Yaskawa INFORM job: X4-SCHODKI_ZEW_HARDOX.JBI

/JOB
//NAME X4-SCHODKI_ZEW_HARDOX
//POS
///NPOS 533,533,533,13,0,0
///TOOL 0
///POSTYPE PULSE
///PULSE
C00000=-21160,-126487,-99095,-6220,53097,-19917
C00001=-122314,-84956,-84267,-5758,65294,-20346
C00002=-113867,-2788,-32259,-11364,77586,20622
C00003=-111699,9606,-11794,-12514,71800,21939
C00004=-110873,16102,-4909,-12893,71047,22311
C00005=-111426,18220,-2948,-12689,70847,22135
C00006=-111334,17863,-3281,-12723,70881,22164
C00007=-111334,17842,-1921,-12786,70054,22254
C00008=-111688,13758,-7042,-12574,71029,22022
C00009=-137921,23655,2193,26065,80546,-13065
C00010=-138187,30095,8478,26164,80127,-13260
C00011=-137141,31636,10013,25924,79665,-12972
C00012=-137283,31426,9804,25956,79727,-13011
C00013=-137283,31447,11085,26011,79025,-13166
C00014=-137811,24810,3269,26040,80453,-13045
C00015=-130093,15204,-5597,17076,73087,-3422
C00016=-130254,16762,-4164,17139,73044,-3486
C00017=-130499,11823,-8660,17205,73314,-3535
C00018=-136657,16032,-4835,19303,74485,-5576
C00019=-136779,34044,12201,19450,73350,-5806
C00020=-136367,37287,16065,19383,72578,-5782
C00021=-135529,38270,17077,19116,72272,-5524
C00022=-135735,38345,17156,19186,72312,-5593
C00023=-135735,38391,18179,19247,71738,-5687
C00024=-136093,38073,17157,19317,72259,-5733
C00025=-136821,38987,18103,19565,72324,-5991
C00026=-137234,41236,20445,19732,72152,-6174
C00027=-137468,37941,16529,19737,72884,-6137
C00028=-139273,33119,8814,10616,74138,-14432
C00029=-138400,39162,15428,10360,73077,-14220
C00030=-137624,40756,17090,10099,72782,-13973
C00031=-137810,40443,16764,10163,72844,-14033
C00032=-137810,40460,18419,10216,71849,-14119
C00033=-138377,33107,10032,10341,73283,-14197
C00034=-129933,32626,9546,-1459,71562,-3103
C00035=-130107,34413,11352,-1398,71367,-3162
C00036=-130344,28976,5916,-1305,71915,-3250
C00037=-134876,30968,7890,396,71698,-4822
C00038=-142592,70732,50995,12851,68399,-16892
C00039=-141830,71409,51797,12602,68137,-16639
C00040=-142006,70894,51186,12652,68274,-16689
C00041=-142006,71149,52557,12712,67578,-16765
C00042=-142006,71007,51815,12679,67954,-16725
C00043=-142747,76515,58410,13043,66871,-17119
C00044=-142702,66110,44987,12780,69711,-16790
C00045=-130401,22900,-3912,-9781,74013,-14096
C00046=-130750,-77898,-76934,-10038,67211,-13654
C00047=-128341,-94500,-64478,-15665,37561,-8814
C00048=-125354,-34494,-33676,-16070,41961,-8103
C00049=-123908,-22688,-35224,7311,60763,-8117
C00050=-115329,1774,-22996,8583,68206,-33205
C00051=-113811,6923,-16554,7934,66753,-32769
C00052=-112938,8598,-15088,7517,66630,-32466
C00053=-113357,7607,-15958,7718,66694,-32611
C00054=-113357,7474,-14642,7767,65823,-32669
C00055=-113357,7562,-15559,7732,66427,-32629
C00056=-114674,8046,-17033,9196,71995,-10105
C00057=-114277,9137,-16073,9034,71921,-9973
C00058=-114994,10710,-14679,9331,71949,-10219
C00059=-115929,5782,-19714,10610,72890,-11247
C00060=-114914,9168,-18033,20160,83408,-25507
C00061=-115077,46309,11834,20851,92481,-23935
C00062=-115077,45981,13257,20825,91503,-24106
C00063=-115077,46309,11834,20851,92481,-23935
C00064=-114509,10430,-16126,20066,82816,-25464
C00065=-113574,12027,-14696,19812,82540,-25184
C00066=-113966,9476,-16971,19916,82715,-25292
C00067=-109617,50730,10299,20838,92897,-21763
C00068=-109849,50897,10058,15384,88802,-23804
C00069=-109890,48745,8449,15106,86687,-24128
C00070=-110280,52401,12404,10304,83703,-19954
C00071=-110340,48514,8983,10012,81065,-20250
C00072=-109875,50139,10594,6927,80049,-17487
C00073=-111642,41129,-2073,7513,83338,-17864
C00074=-120740,-4591,-30289,15267,55452,-23675
C00075=-120758,-111403,-89341,20679,37744,-27189
C00076=-120758,-111403,-89341,20679,37744,-27189
C00077=-97140,-41370,-74515,-11864,90116,15742
C00078=-93918,-16818,-51601,-15265,90472,19448
C00079=-96838,-21310,-54909,-14446,89719,18600
C00080=-97144,-22320,-55662,-14359,89616,18514
C00081=-98771,-24881,-57497,-13895,89173,18041
C00082=-115828,-29996,-61044,7286,86100,-2495
C00083=-121364,-24267,-57094,13933,89260,-9154
C00084=-125064,-13370,-49143,14990,90552,-10191
C00085=-125209,-12228,-48362,15033,90681,-10222
C00086=-127775,-3453,-41245,15747,91251,-10973
C00087=-117906,-11103,-47413,1372,86513,3179
C00088=-107817,-4833,-42392,-13913,90158,17947
C00089=-111065,-8601,-45456,-12965,89620,16971
C00090=-111228,-9142,-45834,-12917,89553,16926
C00091=-113235,-11504,-47787,-12324,89257,16321
C00092=-116129,-16038,-53218,-11461,89860,15351
C00093=-132129,3503,-37461,-731,88042,5165
C00094=-135089,9999,-29918,1559,86605,3002
C00095=-133932,10352,-29664,1179,86614,3356
C00096=-133300,11122,-28999,967,86593,3553
C00097=-132997,13157,-27039,5636,86965,-851
C00098=-131112,-12606,-50888,7793,88905,-29033
C00099=-129834,-10886,-48018,7386,87922,-28697
C00100=-133242,1411,-38107,8469,88444,-29724
C00101=-133268,2556,-37251,8479,88508,-29727
C00102=-132895,14601,-26523,2898,86979,-24450
C00103=-133144,15447,-25750,2979,86944,-24527
C00104=-133588,9909,-35564,3125,90148,-24585
C00105=-114600,-38617,-66572,-24501,76796,-21744
C00106=-88804,-102668,-113384,-34072,81784,-13502
C00107=3643,-76224,-106676,19950,71810,76872
C00108=6047,-95755,-92046,-14751,98253,9605
C00109=8024,-164446,-133802,-16041,6272,12396
C00110=8024,-164446,-133802,-16041,6272,12396
C00111=80911,-131071,-112390,-19160,57527,-4768
C00112=107387,-112645,-89313,-18613,48039,-3448
C00113=120529,-94925,-67119,-18087,38914,-2179
C00114=119158,-22093,-21003,-8683,62714,-5793
C00115=120616,-13235,-11129,-9376,61371,-5124
C00116=120244,-10241,-8815,-9223,61441,-5272
C00117=120242,-11093,-9478,-9225,61411,-5270
C00118=120242,-10458,-7028,-9331,60244,-5174
C00119=120224,-17007,-14555,-9215,61493,-5286
C00120=122889,-18524,910,-53470,54044,-6110
C00121=122847,-15690,3005,-53366,54123,-6195
C00122=122811,-12986,5045,-53281,54183,-6262
C00123=122821,-13724,4484,-53302,54168,-6245
C00124=122821,-12957,6355,-53740,53705,-5906
C00125=125895,-21581,-2992,-53539,56263,-5738
C00126=123923,-36868,-26996,-37261,61302,-5894
C00127=108816,-52753,-53811,-10212,62008,-9374
C00128=96034,-45136,-47055,9675,61622,-25160
C00129=97205,-43220,-45890,9111,61748,-24699
C00130=96974,-43470,-46044,9221,61740,-24787
C00131=96974,-43222,-44278,9303,60791,-24865
C00132=96448,-45521,-47615,9470,61714,-24990
C00133=118629,-40101,-48504,-12157,74776,12413
C00134=119364,-34097,-44083,-12359,75244,12623
C00135=118100,-32224,-42841,-11965,75251,12181
C00136=118253,-32582,-43080,-12015,75236,12237
C00137=118253,-32540,-41664,-12057,74406,12319
C00138=118721,-32602,-42752,-12165,75101,12411
C00139=116137,-37716,-46090,-11401,74165,11593
C00140=108993,-39238,-47060,-3979,71836,3847
C00141=109761,-37600,-46019,-4238,72074,4108
C00142=108993,-39238,-47060,-3979,71836,3847
C00143=117414,-43467,-49690,-6866,71847,6805
C00144=120406,-23125,-36428,-7781,74390,7697
C00145=120412,-21128,-34805,-7781,74419,7698
C00146=119620,-19753,-33804,-7516,74437,7425
C00147=119849,-20298,-34202,-7592,74423,7506
C00148=119849,-20300,-33096,-7616,73750,7551
C00149=119849,-20302,-33703,-7602,74119,7528
C00150=120845,-19874,-33391,-7929,74241,7866
C00151=121446,-18122,-32105,-8123,74405,8066
C00152=121464,-22241,-35587,-8130,74432,8070
C00153=122270,-32243,-42159,4732,69932,24573
C00154=121378,-24903,-37120,5049,70656,24286
C00155=120376,-23507,-36128,5424,70830,23939
C00156=120533,-24190,-36613,5366,70768,23993
C00157=120533,-24175,-35602,5386,70155,23966
C00158=120148,-30314,-42064,5504,71001,23867
C00159=110805,-25383,-38662,15109,74916,14576
C00160=111818,-22665,-36734,14771,74934,14940
C00161=111748,-27369,-40047,14817,74581,14871
C00162=119775,-28434,-40781,12151,73173,17551
C00163=124224,-1084,-19915,10540,73751,19166
C00164=130157,198,-18683,-209,73628,24476
C00165=130157,158,-17341,-210,72780,24477
C00166=130157,185,-18394,-210,73442,24477
C00167=129196,1421,-17357,132,73439,24146
C00168=130157,185,-18394,-210,73442,24477
C00169=122787,3680,-15441,12656,76349,11624
C00170=123743,5439,-13926,12357,76179,11938
C00171=123109,1410,-18093,12531,76759,11776
C00172=126751,-18741,-32489,13679,66636,29547
C00173=131594,-6512,-22252,11541,65879,31250
C00174=135627,-1986,-17513,3780,65616,32121
C00175=134567,7692,-12619,5089,73681,32152
C00176=134567,7658,-11680,5104,73087,32127
C00177=135627,-1986,-17486,3780,65599,32120
C00178=134800,-891,-16582,4152,65645,31822
C00179=135627,-1986,-17486,3780,65599,32120
C00180=122949,-12611,-24589,22132,67603,15841
C00181=121506,-8744,-21577,22663,68115,15387
C00182=122081,-6475,-19773,22437,68011,15585
C00183=121506,-8744,-21577,22663,68115,15387
C00184=127706,-12999,-26066,20142,67056,17565
C00185=135610,17691,-1290,8706,67320,35420
C00186=135610,17711,-348,8741,66754,35378
C00187=136075,11798,-4304,8086,62236,35152
C00188=136366,13707,-2741,6760,62424,35173
C00189=136075,11798,-4304,8086,62236,35152
C00190=131305,-10305,-23416,10361,63176,33430
C00191=168291,-111367,-82610,-9688,47305,48503
C00192=206286,-74639,-65979,-25452,64014,61826
C00193=159660,-110455,-93035,-14572,38895,45711
C00194=139772,-9678,-45421,-20416,66544,-77404
C00195=128522,-26109,-48700,-36268,57340,-84657
C00196=119767,-9340,-33749,-20588,54929,-87055
C00197=118381,-12869,-36453,-19680,54464,-87541
C00198=118069,-13852,-36761,-19540,54093,-87599
C00199=119937,-17804,-39758,-30591,59034,-81437
C00200=119898,-18805,-40392,-30604,58911,-81418
C00201=117451,-25827,-45422,-31757,59099,-80707
C00202=119398,-27349,-44114,-37266,57847,-80053
C00203=122977,-25509,-47564,-34287,62428,-79397
C00204=137466,-21144,-46854,-40649,69913,-75869
C00205=196853,-39310,-56838,-56279,98183,-62272
C00206=239125,-37728,-55833,-56309,98295,-62347
C00207=198880,-64017,-70083,-47949,71692,22240
C00208=95782,-63494,-66422,9583,64100,-25040
C00209=96608,-32442,-40990,7123,69750,-24476
C00210=99153,-41436,-44893,7278,64322,-23821
C00211=98934,-42045,-45261,7777,64334,-23890
C00212=100370,-44106,-46526,7182,63922,-23380
C00213=119741,-40174,-44096,-19149,69535,-259
C00214=121592,-27553,-38534,-18093,79240,10876
C00215=125227,-17250,-31142,-18927,80757,11935
C00216=125393,-15914,-30142,-18963,80861,11977
C00217=127846,-8061,-24015,-19516,81680,12716
C00218=119795,-17677,-31449,-8017,74335,-710
C00219=108325,-15786,-29976,9492,74890,-18554
C00220=111630,-19800,-33189,8434,74445,-17438
C00221=111755,-20573,-33754,8397,74383,-17399
C00222=113687,-22438,-34957,7772,73974,-16756
C00223=117056,-24250,-37509,6639,74313,-15568
C00224=128480,-979,-19969,3779,76440,-7427
C00225=130214,3282,-15364,3237,75722,-6858
C00226=129537,3735,-15090,2864,75741,-6451
C00227=129186,4471,-14460,2975,75747,-6572
C00228=129576,5579,-13546,-2876,75741,-370
C00229=130057,-3886,-22978,-3018,76699,-230
C00230=122913,-28792,-41505,-1480,73376,7564
C00231=125274,-18849,-33719,-4896,77191,17730
C00232=131975,-10313,-25549,-10610,74903,19808
C00233=132069,-9167,-24748,-10635,75011,19832
C00234=135966,6668,-11544,-11862,75556,21141
C00235=130236,2592,-15119,-2350,73160,11427
C00236=128403,-11609,-30449,-1692,75251,10764
C00237=112588,-48510,-57222,11111,73491,6010
C00238=118900,-27089,-23855,-4947,60648,-6067
C00239=130292,-938,239,-22775,68727,4409
C00240=117379,-19874,-3208,-40401,48526,-8648
C00241=111452,-18537,-670,-42583,47269,-4687
C00242=115600,-23691,-9256,-36668,53200,-7502
C00243=123114,-34014,-31898,-14023,63529,-7414
C00244=103776,-61917,-65189,16989,73535,3120
C00245=77625,-115928,-93453,24842,70557,-7280
C00246=80911,-131071,-112390,-19160,57527,-4768
C00247=8024,-164446,-133802,-16041,6272,12396
C00248=8024,-164446,-133802,-16041,6272,12396
C00249=3643,-76224,-106676,19950,71810,76872
C00250=3643,-76224,-106676,19950,71810,76872
C00251=3643,-76224,-106676,19950,71810,76872
C00252=3643,-76224,-106676,19950,71810,76872
C00253=-84926,-80067,-84751,-11816,58952,90735
C00254=-123661,-80067,-84751,-11816,58952,90735
C00255=-122903,-30976,-67088,-11139,71240,89773
C00256=-127139,198,-37668,-8934,68706,88593
C00257=-128438,61784,5096,-11296,104956,84706
C00258=-128499,61338,5461,-11257,104502,84732
C00259=-128499,60609,6014,-11216,103801,84798
C00260=-128499,60703,5938,-11219,103891,84788
C00261=-128273,58374,3262,-11283,104361,84815
C00262=-129063,60229,5392,-11127,103914,84609
C00263=-129975,59592,4657,-10979,103923,84320
C00264=-129063,61136,4723,-11178,104777,84528
C00265=-133608,25580,-26809,3658,85338,86524
C00266=-133451,25659,-25652,3594,84661,86550
C00267=-133451,25176,-25219,3596,84144,86535
C00268=-133451,25290,-25323,3596,84268,86539
C00269=-133704,27427,-23228,3702,84086,86458
C00270=-132883,25504,-25115,3358,84228,86706
C00271=-131959,26058,-24571,2972,84149,86977
C00272=-132883,26390,-25891,3354,85159,86731
C00273=-124009,23376,-33099,9871,93491,73495
C00274=-123836,21523,-31842,9785,91773,73411
C00275=-123836,21007,-31440,9780,91267,73370
C00276=-123836,21118,-31523,9779,91378,73378
C00277=-124020,21136,-31509,9844,91394,73325
C00278=-123836,21717,-31986,9786,91960,73425
C00279=-123362,54647,1396,9599,88337,73286
C00280=-123280,54093,1879,9571,87758,73266
C00281=-123280,53580,2373,9572,87197,73224
C00282=-123280,53684,2271,9572,87311,73232
C00283=-123445,53701,2290,9630,87327,73184
C00284=-123280,54390,1609,9571,88071,73290
C00285=-125487,1894,-47010,15546,81241,73431
C00286=-125038,-918,-46164,15415,79269,73319
C00287=-125038,-1557,-45483,15449,78547,73228
C00288=-125038,-1296,-45768,15435,78846,73266
C00289=-124792,-4958,-48763,15321,78767,73334
C00290=-124792,-5291,-48397,15341,78383,73286
C00291=-124942,-3860,-47236,15411,78431,73246
C00292=-124949,-3247,-48411,15367,79433,73371
C00293=-117766,4954,-42293,11937,78807,75522
C00294=-117765,4385,-41727,11960,78179,75462
C00295=-117765,3691,-40987,11993,77383,75384
C00296=-117765,3905,-41223,11983,77632,75409
C00297=-117315,-1199,-45523,11766,77597,75546
C00298=-117315,-1510,-45179,11782,77233,75510
C00299=-117558,529,-43483,11899,77268,75437
C00300=-117512,138,-43810,11877,77262,75451
C00301=-118420,-299,-44174,12317,77382,75178
C00302=-118236,775,-45287,12178,78567,75353
C00303=-118072,3935,-47958,-6388,83076,70255
C00304=-117672,-3023,-48934,-6614,80148,70526
C00305=-117672,-3736,-48216,-6630,79346,70569
C00306=-117672,-3529,-48430,-6626,79583,70556
C00307=-117228,-8786,-52641,-6836,79506,70694
C00308=-117228,-9038,-52379,-6842,79217,70710
C00309=-117506,-6503,-50372,-6711,79263,70623
C00310=-117501,-5841,-51500,-6695,80291,70569
C00311=-140420,-5323,-52894,-1425,79407,62151
C00312=-145152,-6893,-50667,901,77218,60735
C00313=-145152,-7520,-49981,903,76471,60731
C00314=-145152,-7282,-50248,902,76758,60733
C00315=-145549,-12922,-54644,1100,76568,60610
C00316=-145549,-13251,-54270,1101,76169,60607
C00317=-145357,-10860,-52432,1005,76265,60667
C00318=-145454,-10428,-54083,1049,77503,60647
C00319=-128438,61784,5096,-11296,104956,84706
C00320=-125432,64694,8496,-11765,104746,85676
C00321=-124662,61530,7092,-11845,104102,85987
C00322=-129042,57667,2638,-11155,104293,84576
C00323=-129042,57667,2638,-11155,104293,84576
C00324=-130604,43844,-10848,-9440,96834,84970
C00325=-134320,25640,-25171,-1592,84682,85843
C00326=-137130,19028,-28909,5529,79562,86298
C00327=-133173,20661,-27367,3689,79252,87491
C00328=-133173,20661,-27367,3689,79252,87491
C00329=-130137,46597,-8299,-623,96129,87922
C00330=-124662,61530,7092,-11845,104102,85987
C00331=-124774,62733,6607,-11885,104986,85864
C00332=-124009,23376,-33099,9871,93491,73495
C00333=-124132,1653,-46107,10219,82838,72685
C00334=-124081,891,-45397,10214,82014,72632
C00335=-123957,9856,-37642,10163,81837,72656
C00336=-123957,10397,-38161,10152,82425,72704
C00337=-123328,56859,331,9544,106484,74564
C00338=-123371,55361,-743,9544,106381,74542
C00339=-123850,18974,-31534,9940,86065,72993
C00340=-123271,52328,2620,9755,82174,72867
C00341=-123271,52662,2260,9748,82562,72897
C00342=-127589,85070,34886,10208,94705,72346
C00343=-127605,84117,34810,10205,94272,72304
C00344=-128402,52886,4535,12032,80236,71108
C00345=-128225,58749,11133,11991,79186,71062
C00346=-128225,59756,9915,11950,80426,71182
C00347=-127948,-6468,-52224,16731,80618,72590
C00348=-127424,-2906,-46525,16565,78913,72521
C00349=-130398,-3517,-45707,22203,78529,72642
C00350=-129750,-4200,-46262,21908,78366,72825
C00351=-128378,-4058,-46148,21277,78045,73219
C00352=-121663,-2339,-44741,18114,76618,75175
C00353=-115640,-347,-45187,7560,78187,75189
C00354=-115728,877,-44163,7601,78193,75162
C00355=-120769,-437,-43402,17007,76693,75297
C00356=-117743,897,-42286,15536,76152,76198
C00357=-117743,1848,-43354,15471,77259,76340
C00358=-127948,-6468,-52224,16731,80618,72590
C00359=-117890,-3178,-50858,3,81161,72238
C00360=-118337,-2948,-47894,214,79455,72104
C00361=-118633,-4108,-48842,352,79442,72013
C00362=-119043,-4814,-49224,544,79316,71888
C00363=-117595,-6540,-50048,-6610,79040,70621
C00364=-148660,-7034,-50440,8059,79279,61212
C00365=-144502,-3981,-44897,-14956,77034,56051
C00366=-144502,-3024,-46070,-14896,78209,55905
C00367=-121650,-5019,-58113,-24818,88994,61227
C00368=-122271,-90655,-108273,-25102,76857,63579
C00369=32571,-155976,-119807,-12475,-16322,90735
C00370=32571,-155976,-119807,-12475,-16322,90735
C00371=432,-155976,-119807,-12475,-16322,90735
C00372=432,-155976,-119807,609,74424,82099
C00373=109557,-155976,-119807,609,74424,82099
C00374=131526,-73725,-103845,608,74936,82102
C00375=123676,15402,-35905,4513,79152,79802
C00376=123062,13907,-34117,4846,77322,79548
C00377=123062,13234,-33422,4858,76552,79519
C00378=123062,13371,-33570,4856,76713,79525
C00379=122641,9174,-37336,5063,76896,79403
C00380=122641,8998,-37151,5067,76691,79395
C00381=122935,11565,-34861,4920,76586,79481
C00382=122946,11968,-36957,4889,78077,79544
C00383=128447,74843,20112,4181,96979,82150
C00384=125283,85916,34561,10572,99934,82307
C00385=125283,85252,35263,10543,99176,82240
C00386=125283,85360,35146,10549,99299,82250
C00387=125053,82619,31732,10612,100007,82237
C00388=130133,63218,10337,-478,91768,81983
C00389=129424,63758,10966,-266,91655,81768
C00390=130133,64176,9529,-479,92758,81979
C00391=130562,33088,-16638,4936,77416,83764
C00392=130793,32566,-15857,4835,76660,83805
C00393=130793,32167,-15406,4840,76179,83784
C00394=130793,32267,-15524,4840,76302,83790
C00395=131028,34733,-13015,4729,76015,83854
C00396=131220,32098,-15696,4631,76299,83921
C00397=132054,31571,-16260,4222,76334,84182
C00398=131220,33089,-16758,4612,77459,83964
C00399=139932,37494,-12236,353,76701,86621
C00400=140087,35879,-12490,279,76027,86666
C00401=140087,35493,-12044,279,75554,86665
C00402=140087,35594,-12164,279,75679,86665
C00403=140066,35120,-12650,289,75735,86658
C00404=140191,35640,-13057,228,76251,86698
C00405=144017,27791,-20964,-1648,77113,87870
C00406=144452,26542,-22051,-1859,77149,88000
C00407=144452,26082,-21554,-1861,76609,88006
C00408=144452,26191,-21674,-1860,76739,88004
C00409=144404,25656,-22195,-1836,76786,87989
C00410=144440,26768,-22186,-1850,77351,87992
C00411=131883,61278,7206,30840,98791,74831
C00412=134379,62597,12993,30002,95475,74827
C00413=134379,61982,13733,29953,94803,74651
C00414=134379,62041,13659,29957,94869,74668
C00415=134641,60677,12085,29912,95014,74800
C00416=134557,61287,11866,29960,95432,74879
C00417=135751,64817,15957,29630,94430,75042
C00418=135751,64366,16527,29599,93921,74910
C00419=135751,64464,16397,29606,94034,74940
C00420=136038,63706,15517,29546,94076,75054
C00421=135884,64035,14878,29615,94618,75138
C00422=132248,54311,3772,30620,97400,74580
C00423=132248,53898,4219,30579,96978,74466
C00424=132248,54015,4093,30592,97096,74498
C00425=129743,23890,-20564,36987,85720,58400
C00426=129743,23766,-20396,36992,85584,58355
C00427=129558,27733,-16530,37067,85382,58218
C00428=129612,27679,-19165,37009,86646,58668
C00429=128447,74843,20112,4181,96979,82150
C00430=123342,73095,22025,-160,83462,78859
C00431=123154,73616,24314,-89,82322,78803
C00432=123153,73142,24904,-89,81719,78803
C00433=123153,73214,24808,-89,81815,78803
C00434=123322,73233,24831,-152,81812,78855
C00435=123242,73796,24123,-122,82537,78829
C00436=123688,38124,-16975,-287,89497,78950
C00437=123584,37405,-16446,-248,88799,78920
C00438=123584,36852,-15992,-248,88235,78921
C00439=123584,36953,-16076,-248,88338,78921
C00440=123771,37027,-15999,-318,88331,78976
C00441=123711,37942,-16737,-296,89256,78956
C00442=125600,30882,-21833,-7436,86676,77848
C00443=125600,30421,-21439,-7437,86203,77876
C00444=125600,30651,-21637,-7436,86441,77862
C00445=125408,25580,-26659,-7358,86908,77778
C00446=125408,25321,-26441,-7359,86643,77794
C00447=125473,27805,-24002,-7386,86425,77827
C00448=125473,28768,-24793,-7383,87400,77770
C00449=119735,35798,-17668,-5085,86249,76136
C00450=119539,34421,-18220,-5006,85875,76095
C00451=119539,33880,-17746,-5008,85308,76118
C00452=119539,34054,-17902,-5007,85493,76110
C00453=119038,29010,-22988,-4803,86002,75940
C00454=119038,28800,-22804,-4803,85784,75950
C00455=119400,31604,-19998,-4950,85517,76067
C00456=119348,31196,-20409,-4929,85557,76050
C00457=119987,30698,-20909,-5185,85643,76236
C00458=119878,31262,-21389,-5139,86220,76180
C00459=128447,74843,20112,4181,96979,82150
C00460=124116,94593,46679,11672,102200,82046
C00461=127992,89556,40269,11396,103012,83415
C00462=127992,89556,40269,11396,103012,83415
C00463=129587,64527,11769,9334,94236,82902
C00464=132949,55867,3405,1789,88718,82304
C00465=135017,42183,-7617,-3983,80598,81730
C00466=131389,44285,-5377,-2395,80172,80630
C00467=131389,44285,-5377,-2395,80172,80630
C00468=132236,58768,6599,-5557,89172,80111
C00469=124116,94593,46679,11672,102200,82046
C00470=124104,96699,46972,11722,103085,82128
C00471=143616,55927,3157,-10764,85977,88488
C00472=148648,52226,4712,-20280,79209,89000
C00473=148516,52517,6145,-20267,78491,89078
C00474=148493,50806,4254,-20239,78754,89026
C00475=148493,50806,4254,-20239,78754,89026
C00476=140540,62715,11224,-1744,88121,79582
C00477=136875,97884,50516,6622,100207,80085
C00478=137178,101903,55708,7300,101861,80376
C00479=141388,85873,34619,7196,106210,82037
C00480=141388,85873,34619,7196,106210,82037
C00481=144251,72599,18557,4985,103495,82483
C00482=142808,65433,11761,11663,99026,82997
C00483=143036,65995,12421,11611,98881,83056
C00484=141225,66295,15146,18784,94862,83443
C00485=141225,67539,13983,18842,96148,83643
C00486=134946,24098,-37413,1605,94871,78009
C00487=119914,5828,-43406,7387,78039,72896
C00488=119947,11480,-35472,7422,76073,72788
C00489=122612,12239,-33354,1270,74705,81494
C00490=122593,20325,-25822,1280,74225,81483
C00491=122593,20926,-26500,1276,74951,81491
C00492=122252,68374,13418,1881,98899,81800
C00493=122183,71569,17944,1970,100800,81820
C00494=122504,26900,-20597,1350,76261,81486
C00495=122262,60388,15081,1504,71520,81353
C00496=122262,60839,14399,1498,72171,81361
C00497=122138,113341,70542,1866,86603,81577
C00498=122006,122876,83892,1956,86819,81545
C00499=122146,80790,34625,1654,78685,81435
C00500=122106,87009,42344,1679,77132,81400
C00501=122106,87849,40937,1672,78429,81417
C00502=119914,5828,-43406,7387,78039,72896
C00503=119947,11480,-35472,7422,76073,72788
C00504=127628,12770,-32579,-8395,74956,81127
C00505=127315,11373,-33838,-8234,74983,81029
C00506=128071,4553,-37059,-10767,69794,81127
C00507=127715,4566,-37046,-10566,69753,81013
C00508=126468,4857,-36794,-9866,69606,80617
C00509=120231,6674,-35162,-6323,68971,78621
C00510=109035,9040,-32856,15253,70226,79190
C00511=109194,10411,-31638,15171,70156,79234
C00512=119176,8835,-33361,-5116,68948,78440
C00513=122835,8933,-31103,-15912,67286,77485
C00514=123391,8334,-34505,-16043,69107,77423
C00515=119914,5828,-43406,7387,78039,72896
C00516=119947,11480,-35472,7422,76073,72788
C00517=113441,11557,-31162,19125,73394,81975
C00518=113492,10653,-31972,19096,73415,81995
C00519=113877,9453,-33080,18895,73400,82121
C00520=114196,9069,-33420,18732,73346,82217
C00521=115691,8179,-34205,17966,73067,82671
C00522=137435,5926,-34612,18335,69915,81720
C00523=144315,10126,-28780,22360,67559,86040
C00524=145057,10570,-28384,21951,67362,86265
C00525=145057,11493,-29866,21752,68653,86515
C00526=125202,6402,-41617,3278,75462,76453
C00527=131548,-138252,-117845,-124,47939,78402
C00528=-918,-163100,-132191,-124,47939,78402
C00529=-918,-163100,-132191,-124,-6868,78402
C00530=-918,-163100,-132191,-124,-6868,78402
C00531=-918,-163100,-132191,-124,-6868,78402
C00532=-918,-163100,-132191,-124,-6868,78402
BC00000=277659,673923,172124
BC00001=328197,693320,172124
BC00002=328196,693321,172121
BC00003=328196,693321,172121
BC00004=328196,693321,172121
BC00005=328196,693321,172121
BC00006=328196,693321,172121
BC00007=328196,693321,172121
BC00008=328196,693321,172121
BC00009=328196,693321,172121
BC00010=328196,693321,172121
BC00011=328196,693321,172121
BC00012=328196,693321,172121
BC00013=328196,693321,172121
BC00014=328196,693321,172121
BC00015=328196,693321,172121
BC00016=328196,693321,172121
BC00017=328196,693321,172121
BC00018=328196,693321,172121
BC00019=328196,693321,172121
BC00020=328196,693321,172121
BC00021=328196,693321,172121
BC00022=328196,693321,172121
BC00023=328196,693321,172121
BC00024=328196,693321,172121
BC00025=328196,693321,172121
BC00026=328196,693321,172121
BC00027=328196,693321,172121
BC00028=328196,693321,172121
BC00029=328196,693321,172121
BC00030=328196,693321,172121
BC00031=328196,693321,172121
BC00032=328196,693321,172121
BC00033=328196,693321,172121
BC00034=328196,693321,172121
BC00035=328196,693321,172121
BC00036=328196,693321,172121
BC00037=328196,693321,172121
BC00038=328196,693321,172121
BC00039=328196,693321,172121
BC00040=328196,693321,172121
BC00041=328196,693321,172121
BC00042=328196,693321,172121
BC00043=328196,693321,172121
BC00044=328196,693321,172121
BC00045=328196,693321,172121
BC00046=328196,693321,172121
BC00047=194432,688081,172121
BC00048=194432,688081,172121
BC00049=173327,765103,172121
BC00050=173327,765103,140855
BC00051=173327,765103,140855
BC00052=173327,765103,140855
BC00053=173327,765103,140855
BC00054=173327,765103,140855
BC00055=173327,765103,140855
BC00056=173327,765103,140855
BC00057=173327,765103,140855
BC00058=173327,765103,140855
BC00059=173327,765103,140855
BC00060=173327,765103,140855
BC00061=173327,744937,115517
BC00062=173327,744937,115517
BC00063=173327,744937,115517
BC00064=173327,765103,140855
BC00065=173327,765103,140855
BC00066=173327,765103,140855
BC00067=158508,737843,59363
BC00068=158508,737843,59363
BC00069=158508,737843,59363
BC00070=158508,737843,59363
BC00071=158508,737843,59363
BC00072=158508,737843,59363
BC00073=158508,737843,59363
BC00074=158508,737843,59363
BC00075=158508,682152,59363
BC00076=293322,682152,59363
BC00077=293321,752433,59360
BC00078=293321,752433,59360
BC00079=293321,752433,59360
BC00080=293321,752433,59360
BC00081=293321,752433,59360
BC00082=293321,752433,59360
BC00083=293321,752433,59360
BC00084=293321,752433,59360
BC00085=293321,752433,59360
BC00086=293321,752433,59360
BC00087=293321,752433,59360
BC00088=293321,752433,59360
BC00089=293321,752433,59360
BC00090=293321,752433,59360
BC00091=293321,752433,59360
BC00092=293321,752433,59360
BC00093=293321,752433,59360
BC00094=293321,752433,59360
BC00095=293321,752433,59360
BC00096=293321,752433,59360
BC00097=293321,752433,59360
BC00098=293321,752433,59360
BC00099=293321,752433,59360
BC00100=293321,752433,59360
BC00101=293321,752433,59360
BC00102=293321,752433,59360
BC00103=293321,752433,59360
BC00104=293321,752433,59360
BC00105=293321,752433,59360
BC00106=293321,698561,59360
BC00107=199464,674570,1075173
BC00108=95044,675039,919146
BC00109=95044,675039,1075229
BC00110=235813,1345575,1075229
BC00111=291733,1363613,501241
BC00112=295042,1365829,344881
BC00113=288108,1367960,194507
BC00114=288108,1367960,194507
BC00115=288108,1367960,194507
BC00116=288108,1367960,194507
BC00117=288108,1367960,194507
BC00118=288108,1367960,194507
BC00119=288108,1367960,194507
BC00120=288108,1367960,194507
BC00121=288108,1367960,194507
BC00122=288108,1367960,194507
BC00123=288108,1367960,194507
BC00124=288108,1367960,194507
BC00125=288108,1367960,194507
BC00126=288108,1367445,194507
BC00127=288108,1366688,194507
BC00128=288109,1366690,194504
BC00129=288109,1366690,194504
BC00130=288109,1366690,194504
BC00131=288109,1366690,194504
BC00132=288109,1366690,194504
BC00133=288109,1366690,194504
BC00134=288109,1366690,194504
BC00135=288109,1366690,194504
BC00136=288109,1366690,194504
BC00137=288109,1366690,194504
BC00138=288109,1366690,194504
BC00139=288109,1366690,194504
BC00140=288109,1366690,194504
BC00141=288109,1366690,194504
BC00142=288109,1366690,194504
BC00143=288109,1366690,194504
BC00144=288109,1366690,194504
BC00145=288109,1366690,194504
BC00146=288109,1366690,194504
BC00147=288109,1366690,194504
BC00148=288109,1366690,194504
BC00149=288109,1366690,194504
BC00150=288109,1366690,194504
BC00151=288109,1366690,194504
BC00152=288109,1366690,194504
BC00153=288109,1366690,194504
BC00154=288109,1366690,194504
BC00155=288109,1366690,194504
BC00156=288109,1366690,194504
BC00157=288109,1366690,194504
BC00158=288109,1366690,194504
BC00159=288109,1366690,194504
BC00160=288109,1366690,194504
BC00161=288109,1366690,194504
BC00162=288109,1366690,194504
BC00163=288109,1366690,194504
BC00164=288109,1366690,194504
BC00165=288109,1366690,194504
BC00166=288109,1366690,194504
BC00167=288109,1366690,194504
BC00168=288109,1366690,194504
BC00169=288109,1366690,194504
BC00170=288109,1366690,194504
BC00171=288109,1366690,194504
BC00172=288109,1366690,194504
BC00173=288109,1366690,194504
BC00174=288109,1366690,194504
BC00175=288109,1366690,194504
BC00176=288109,1366690,194504
BC00177=288109,1366690,194504
BC00178=288109,1366690,194504
BC00179=288109,1366690,194504
BC00180=288109,1366690,194504
BC00181=288109,1366690,194504
BC00182=288109,1366690,194504
BC00183=288109,1366690,194504
BC00184=288109,1366690,194504
BC00185=288109,1366690,194504
BC00186=288109,1366690,194504
BC00187=288109,1366690,194504
BC00188=288109,1366690,194504
BC00189=288109,1366690,194504
BC00190=288109,1366690,194504
BC00191=362373,1366690,194504
BC00192=212912,1366690,52238
BC00193=212912,1366690,52238
BC00194=212912,1366690,52238
BC00195=181372,1351458,52238
BC00196=181372,1351458,52238
BC00197=181372,1351458,52238
BC00198=181372,1351458,52238
BC00199=181372,1351458,52238
BC00200=181372,1351458,52238
BC00201=181372,1351458,52238
BC00202=181372,1351458,52238
BC00203=181372,1351458,52238
BC00204=181372,1351458,52238
BC00205=258948,1351458,52238
BC00206=397724,1351458,84656
BC00207=397724,1351458,84656
BC00208=288109,1366690,194504
BC00209=288109,1366690,194504
BC00210=288109,1366690,194504
BC00211=288109,1366690,194504
BC00212=288109,1366690,194504
BC00213=288109,1366690,194504
BC00214=288109,1366690,194504
BC00215=288109,1366690,194504
BC00216=288109,1366690,194504
BC00217=288109,1366690,194504
BC00218=288109,1366690,194504
BC00219=288109,1366690,194504
BC00220=288109,1366690,194504
BC00221=288109,1366690,194504
BC00222=288109,1366690,194504
BC00223=288109,1366690,194504
BC00224=288109,1366690,194504
BC00225=288109,1366690,194504
BC00226=288109,1366690,194504
BC00227=288109,1366690,194504
BC00228=288109,1366690,194504
BC00229=288109,1366690,194504
BC00230=288109,1366690,194504
BC00231=288109,1366690,194504
BC00232=288109,1366690,194504
BC00233=288109,1366690,194504
BC00234=288109,1366690,194504
BC00235=288109,1366690,194504
BC00236=288109,1366690,194504
BC00237=288109,1366690,194504
BC00238=288109,1366690,194504
BC00239=288109,1366690,194504
BC00240=288109,1366690,194504
BC00241=288109,1366690,194504
BC00242=288109,1366690,194504
BC00243=288109,1366690,194504
BC00244=288109,1366690,194504
BC00245=288109,1366690,194504
BC00246=269895,1363613,501241
BC00247=235813,1345575,1075229
BC00248=95044,675039,1075229
BC00249=199464,674570,1075173
BC00250=199464,674570,1075173
BC00251=199464,674570,1075173
BC00252=199464,674570,1075173
BC00253=275760,675148,198531
BC00254=313005,675148,45896
BC00255=313005,783706,45896
BC00256=313005,783706,45896
BC00257=323528,783706,0
BC00258=323528,783706,0
BC00259=323528,783706,0
BC00260=323528,783706,0
BC00261=323528,783706,0
BC00262=323528,783706,0
BC00263=323528,783706,0
BC00264=323528,783706,0
BC00265=323528,783706,0
BC00266=323528,783706,0
BC00267=323528,783706,0
BC00268=323528,783706,0
BC00269=323528,783706,0
BC00270=323528,783706,0
BC00271=323528,783706,0
BC00272=323528,783706,0
BC00273=309005,783706,0
BC00274=309005,783706,0
BC00275=309005,783706,0
BC00276=309005,783706,0
BC00277=309005,783706,0
BC00278=309005,783706,0
BC00279=309005,783706,0
BC00280=309005,783706,0
BC00281=309005,783706,0
BC00282=309005,783706,0
BC00283=309005,783706,0
BC00284=309005,783706,0
BC00285=309005,783706,0
BC00286=309005,783706,0
BC00287=309005,783706,0
BC00288=309005,783706,0
BC00289=309005,783706,0
BC00290=309005,783706,0
BC00291=309005,783706,0
BC00292=309005,783706,0
BC00293=309005,783706,0
BC00294=309005,783706,0
BC00295=309005,783706,0
BC00296=309005,783706,0
BC00297=309005,783706,0
BC00298=309005,783706,0
BC00299=309005,783706,0
BC00300=309005,783706,0
BC00301=309005,783706,0
BC00302=309005,783706,0
BC00303=309005,783706,0
BC00304=309005,783706,0
BC00305=309005,783706,0
BC00306=309005,783706,0
BC00307=309005,783706,0
BC00308=309005,783706,0
BC00309=309005,783706,0
BC00310=309005,783706,0
BC00311=309005,783706,0
BC00312=309005,783706,0
BC00313=309005,783706,0
BC00314=309005,783706,0
BC00315=309005,783706,0
BC00316=309005,783706,0
BC00317=309005,783706,0
BC00318=309005,783706,0
BC00319=323528,783706,0
BC00320=323528,783706,0
BC00321=323528,783706,0
BC00322=323528,783706,0
BC00323=323528,783706,0
BC00324=323528,783706,0
BC00325=323528,783706,0
BC00326=323528,783706,0
BC00327=323528,783706,0
BC00328=323528,783706,0
BC00329=323528,783706,0
BC00330=323528,783706,0
BC00331=323528,783706,0
BC00332=309005,783706,0
BC00333=309005,783706,0
BC00334=309005,783706,0
BC00335=309005,783706,0
BC00336=309005,783706,0
BC00337=309005,783706,0
BC00338=309005,783706,0
BC00339=309005,783706,0
BC00340=309005,783706,0
BC00341=309005,783706,0
BC00342=325808,783706,0
BC00343=325808,783706,0
BC00344=325808,783706,0
BC00345=325808,783706,0
BC00346=325808,783706,0
BC00347=309005,783706,0
BC00348=309005,783706,0
BC00349=309005,783706,0
BC00350=309005,783706,0
BC00351=309005,783706,0
BC00352=309005,783706,0
BC00353=309005,783706,0
BC00354=309005,783706,0
BC00355=309005,783706,0
BC00356=309005,783706,0
BC00357=309005,783706,0
BC00358=309005,783706,0
BC00359=309005,783706,0
BC00360=309005,783706,0
BC00361=309005,783706,0
BC00362=309005,783706,0
BC00363=309005,783706,0
BC00364=309005,783706,0
BC00365=309005,783706,0
BC00366=309005,783706,0
BC00367=309005,783706,0
BC00368=309005,664227,0
BC00369=17910,675148,1075141
BC00370=17910,675148,1075141
BC00371=17910,1317205,1075141
BC00372=323892,1317205,1075141
BC00373=323892,1346382,668441
BC00374=323892,1361704,68
BC00375=323892,1361702,64
BC00376=323892,1361702,64
BC00377=323892,1361702,64
BC00378=323892,1361702,64
BC00379=323892,1361702,64
BC00380=323892,1361702,64
BC00381=323892,1361702,64
BC00382=323892,1361702,64
BC00383=323892,1361702,64
BC00384=323892,1361702,64
BC00385=323892,1361702,64
BC00386=323892,1361702,64
BC00387=323892,1361702,64
BC00388=323892,1361702,64
BC00389=323892,1361702,64
BC00390=323892,1361702,64
BC00391=323892,1361702,64
BC00392=323892,1361702,64
BC00393=323892,1361702,64
BC00394=323892,1361702,64
BC00395=323892,1361702,64
BC00396=323892,1361702,64
BC00397=323892,1361702,64
BC00398=323892,1361702,64
BC00399=323892,1361702,64
BC00400=323892,1361702,64
BC00401=323892,1361702,64
BC00402=323892,1361702,64
BC00403=323892,1361702,64
BC00404=323892,1361702,64
BC00405=323892,1361702,64
BC00406=323892,1361702,64
BC00407=323892,1361702,64
BC00408=323892,1361702,64
BC00409=323892,1361702,64
BC00410=323892,1361702,64
BC00411=323892,1361702,64
BC00412=323892,1361702,64
BC00413=323892,1361702,64
BC00414=323892,1361702,64
BC00415=323892,1361702,64
BC00416=323892,1361702,64
BC00417=323892,1361702,64
BC00418=323892,1361702,64
BC00419=323892,1361702,64
BC00420=323892,1361702,64
BC00421=323892,1361702,64
BC00422=323892,1361702,64
BC00423=323892,1361702,64
BC00424=323892,1361702,64
BC00425=323892,1361702,64
BC00426=323892,1361702,64
BC00427=323892,1361702,64
BC00428=323892,1361702,64
BC00429=323892,1361702,64
BC00430=323892,1361702,64
BC00431=323892,1361702,64
BC00432=323892,1361702,63
BC00433=323892,1361702,63
BC00434=323892,1361702,63
BC00435=323892,1361702,63
BC00436=323892,1361702,63
BC00437=323892,1361702,63
BC00438=323892,1361702,63
BC00439=323892,1361702,63
BC00440=323892,1361702,63
BC00441=323892,1361702,63
BC00442=323892,1361702,63
BC00443=323892,1361702,63
BC00444=323892,1361702,63
BC00445=323892,1361702,63
BC00446=323892,1361702,63
BC00447=323892,1361702,63
BC00448=323892,1361702,63
BC00449=323892,1361702,63
BC00450=323892,1361702,63
BC00451=323892,1361702,63
BC00452=323892,1361702,63
BC00453=323892,1361702,63
BC00454=323892,1361702,63
BC00455=323892,1361702,63
BC00456=323892,1361702,63
BC00457=323892,1361702,63
BC00458=323892,1361702,63
BC00459=323892,1361702,64
BC00460=323892,1361702,64
BC00461=323892,1361702,64
BC00462=323892,1361702,64
BC00463=323892,1361702,64
BC00464=323892,1361702,64
BC00465=323892,1361702,64
BC00466=323892,1361702,64
BC00467=323892,1361702,64
BC00468=323892,1361702,64
BC00469=323892,1361702,64
BC00470=323892,1361702,64
BC00471=323892,1361702,64
BC00472=323892,1361702,64
BC00473=323892,1361702,64
BC00474=323892,1361702,64
BC00475=323892,1361702,64
BC00476=323892,1361702,63
BC00477=323892,1361702,63
BC00478=323892,1361702,63
BC00479=323892,1361702,63
BC00480=323892,1361702,63
BC00481=323892,1361702,63
BC00482=323892,1361702,63
BC00483=323892,1361702,63
BC00484=323892,1361702,63
BC00485=323892,1361702,63
BC00486=323892,1361702,63
BC00487=323892,1361702,63
BC00488=323892,1361702,63
BC00489=323892,1361702,63
BC00490=323892,1361702,63
BC00491=323892,1361702,63
BC00492=323892,1361702,63
BC00493=323892,1361702,63
BC00494=323892,1361702,63
BC00495=323892,1361702,63
BC00496=323892,1361702,63
BC00497=323892,1361702,63
BC00498=323892,1361702,63
BC00499=323892,1361702,63
BC00500=323892,1361702,63
BC00501=323892,1361702,63
BC00502=323892,1361702,63
BC00503=323892,1361702,63
BC00504=323892,1361702,63
BC00505=323892,1361702,63
BC00506=323892,1361702,63
BC00507=323892,1361702,63
BC00508=323892,1361702,63
BC00509=323892,1361702,63
BC00510=323892,1361702,63
BC00511=323892,1361702,63
BC00512=323892,1361702,63
BC00513=323892,1361702,63
BC00514=323892,1361702,63
BC00515=323892,1361702,63
BC00516=323892,1361702,63
BC00517=323892,1361702,63
BC00518=323892,1361702,63
BC00519=323892,1361702,62
BC00520=323892,1361702,62
BC00521=323892,1361702,62
BC00522=323892,1361702,62
BC00523=323892,1361702,61
BC00524=323892,1361702,61
BC00525=323892,1361702,61
BC00526=323892,1361702,63
BC00527=323892,1361702,62
BC00528=323892,1361702,62
BC00529=323892,1361702,540287
BC00530=266401,1307423,1031512
BC00531=107680,1169688,1031512
BC00532=107680,692424,1031512
EC00000=-798156,0
EC00001=-798156,0
EC00002=-798153,-1
EC00003=-798153,-1
EC00004=-798153,-1
EC00005=-798153,-1
EC00006=-798153,-1
EC00007=-798153,-1
EC00008=-798153,-1
EC00009=-798153,-1
EC00010=-798153,-1
EC00011=-798153,-1
EC00012=-798153,-1
EC00013=-798153,-1
EC00014=-798153,-1
EC00015=-798153,-1
EC00016=-798153,-1
EC00017=-798153,-1
EC00018=-798153,-1
EC00019=-798153,-1
EC00020=-798153,-1
EC00021=-798153,-1
EC00022=-798153,-1
EC00023=-798153,-1
EC00024=-798153,-1
EC00025=-798153,-1
EC00026=-798153,-1
EC00027=-798153,-1
EC00028=-798153,-1
EC00029=-798153,-1
EC00030=-798153,-1
EC00031=-798153,-1
EC00032=-798153,-1
EC00033=-798153,-1
EC00034=-798153,-1
EC00035=-798153,-1
EC00036=-798153,-1
EC00037=-798153,-1
EC00038=-798153,-1
EC00039=-798153,-1
EC00040=-798153,-1
EC00041=-798153,-1
EC00042=-798153,-1
EC00043=-798153,-1
EC00044=-798153,-1
EC00045=-798153,-1
EC00046=-798153,-1
EC00047=-798153,-1
EC00048=-798153,-1
EC00049=-798153,-1
EC00050=-798153,-1
EC00051=-798153,-1
EC00052=-798153,-1
EC00053=-798153,-1
EC00054=-798153,-1
EC00055=-798153,-1
EC00056=-798153,-1
EC00057=-798153,-1
EC00058=-798153,-1
EC00059=-798153,-1
EC00060=-798153,-1
EC00061=-798153,-1
EC00062=-798153,-1
EC00063=-798153,-1
EC00064=-798153,-1
EC00065=-798153,-1
EC00066=-798153,-1
EC00067=-798153,-1
EC00068=-798153,-1
EC00069=-798153,-1
EC00070=-798153,-1
EC00071=-798153,-1
EC00072=-798153,-1
EC00073=-798153,-1
EC00074=-798153,-1
EC00075=-798153,-1
EC00076=-798153,-1
EC00077=-798151,-2
EC00078=-798151,-2
EC00079=-798151,-2
EC00080=-798151,-2
EC00081=-798151,-2
EC00082=-798151,-2
EC00083=-798151,-2
EC00084=-798151,-2
EC00085=-798151,-2
EC00086=-798151,-2
EC00087=-798151,-2
EC00088=-798151,-2
EC00089=-798151,-2
EC00090=-798151,-2
EC00091=-798151,-2
EC00092=-798151,-2
EC00093=-798151,-2
EC00094=-798151,-2
EC00095=-798151,-2
EC00096=-798151,-2
EC00097=-798151,-2
EC00098=-798151,-2
EC00099=-798151,-2
EC00100=-798151,-2
EC00101=-798151,-2
EC00102=-798151,-2
EC00103=-798151,-2
EC00104=-798151,-2
EC00105=-798151,-2
EC00106=-798151,-2
EC00107=-798151,-2
EC00108=-798156,0
EC00109=798156,0
EC00110=798156,0
EC00111=798156,0
EC00112=798156,0
EC00113=798156,0
EC00114=798156,0
EC00115=798156,0
EC00116=798156,0
EC00117=798156,0
EC00118=798156,0
EC00119=798156,0
EC00120=798156,0
EC00121=798156,0
EC00122=798156,0
EC00123=798156,0
EC00124=798156,0
EC00125=798156,0
EC00126=798156,0
EC00127=798156,0
EC00128=798155,0
EC00129=798155,0
EC00130=798155,0
EC00131=798155,0
EC00132=798155,0
EC00133=798155,0
EC00134=798155,0
EC00135=798155,0
EC00136=798155,0
EC00137=798155,0
EC00138=798155,0
EC00139=798155,0
EC00140=798155,0
EC00141=798155,0
EC00142=798155,0
EC00143=798155,0
EC00144=798155,0
EC00145=798155,0
EC00146=798155,0
EC00147=798155,0
EC00148=798155,0
EC00149=798155,0
EC00150=798155,0
EC00151=798155,0
EC00152=798155,0
EC00153=798155,0
EC00154=798155,0
EC00155=798155,0
EC00156=798155,0
EC00157=798155,0
EC00158=798155,0
EC00159=798155,0
EC00160=798155,0
EC00161=798155,0
EC00162=798155,0
EC00163=798155,0
EC00164=798155,0
EC00165=798155,0
EC00166=798155,0
EC00167=798155,0
EC00168=798155,0
EC00169=798155,0
EC00170=798155,0
EC00171=798155,0
EC00172=798155,0
EC00173=798155,0
EC00174=798155,0
EC00175=798155,0
EC00176=798155,0
EC00177=798155,0
EC00178=798155,0
EC00179=798155,0
EC00180=798155,0
EC00181=798155,0
EC00182=798155,0
EC00183=798155,0
EC00184=798155,0
EC00185=798155,0
EC00186=798155,0
EC00187=798155,0
EC00188=798155,0
EC00189=798155,0
EC00190=798155,0
EC00191=798155,0
EC00192=798155,0
EC00193=798155,0
EC00194=798155,0
EC00195=798155,0
EC00196=798155,0
EC00197=798155,0
EC00198=798155,0
EC00199=798155,0
EC00200=798155,0
EC00201=798155,0
EC00202=798155,0
EC00203=798155,0
EC00204=798155,0
EC00205=798155,0
EC00206=798155,0
EC00207=798155,0
EC00208=798155,0
EC00209=798155,0
EC00210=798155,0
EC00211=798155,0
EC00212=798155,0
EC00213=798155,0
EC00214=798155,0
EC00215=798155,0
EC00216=798155,0
EC00217=798155,0
EC00218=798155,0
EC00219=798155,0
EC00220=798155,0
EC00221=798155,0
EC00222=798155,0
EC00223=798155,0
EC00224=798155,0
EC00225=798155,0
EC00226=798155,0
EC00227=798155,0
EC00228=798155,0
EC00229=798155,0
EC00230=798155,0
EC00231=798155,0
EC00232=798155,0
EC00233=798155,0
EC00234=798155,0
EC00235=798155,0
EC00236=798155,0
EC00237=798155,0
EC00238=798155,0
EC00239=798155,0
EC00240=798155,0
EC00241=798155,0
EC00242=798155,0
EC00243=798155,0
EC00244=798155,0
EC00245=798155,0
EC00246=798156,0
EC00247=798156,0
EC00248=798156,0
EC00249=798156,0
EC00250=1521,567
EC00251=0,1112952
EC00252=-798157,1112952
EC00253=-798157,1112952
EC00254=-798157,1112952
EC00255=-798157,1112952
EC00256=-798157,1112952
EC00257=-798156,1112952
EC00258=-798156,1112952
EC00259=-798156,1112952
EC00260=-798156,1112952
EC00261=-798156,1112952
EC00262=-798156,1112952
EC00263=-798156,1112952
EC00264=-798156,1112952
EC00265=-798156,1112952
EC00266=-798156,1112952
EC00267=-798156,1112952
EC00268=-798156,1112952
EC00269=-798156,1112952
EC00270=-798156,1112952
EC00271=-798156,1112952
EC00272=-798156,1112952
EC00273=-798156,1112952
EC00274=-798156,1112952
EC00275=-798156,1112952
EC00276=-798156,1112952
EC00277=-798156,1112952
EC00278=-798156,1112952
EC00279=-798156,1112952
EC00280=-798156,1112952
EC00281=-798156,1112952
EC00282=-798156,1112952
EC00283=-798156,1112952
EC00284=-798156,1112952
EC00285=-798156,1112952
EC00286=-798156,1112952
EC00287=-798156,1112952
EC00288=-798156,1112952
EC00289=-798156,1112952
EC00290=-798156,1112952
EC00291=-798156,1112952
EC00292=-798156,1112952
EC00293=-798156,1112952
EC00294=-798156,1112952
EC00295=-798156,1112952
EC00296=-798156,1112952
EC00297=-798156,1112952
EC00298=-798156,1112952
EC00299=-798156,1112952
EC00300=-798156,1112952
EC00301=-798156,1112952
EC00302=-798156,1112952
EC00303=-798156,1112952
EC00304=-798156,1112952
EC00305=-798156,1112952
EC00306=-798156,1112952
EC00307=-798156,1112952
EC00308=-798156,1112952
EC00309=-798156,1112952
EC00310=-798156,1112952
EC00311=-798156,1112952
EC00312=-798156,1112952
EC00313=-798156,1112952
EC00314=-798156,1112952
EC00315=-798156,1112952
EC00316=-798156,1112952
EC00317=-798156,1112952
EC00318=-798156,1112952
EC00319=-798156,1112952
EC00320=-798156,1112952
EC00321=-798156,1112952
EC00322=-798156,1112952
EC00323=-798156,1112952
EC00324=-798156,1112952
EC00325=-798156,1112952
EC00326=-798156,1112952
EC00327=-798156,1112952
EC00328=-798156,1112952
EC00329=-798156,1112952
EC00330=-798156,1112952
EC00331=-798156,1112952
EC00332=-798156,1112952
EC00333=-798156,1112952
EC00334=-798156,1112952
EC00335=-798156,1112952
EC00336=-798156,1112952
EC00337=-798156,1112952
EC00338=-798156,1112952
EC00339=-798156,1112952
EC00340=-798156,1112952
EC00341=-798156,1112952
EC00342=-798156,1112952
EC00343=-798156,1112952
EC00344=-798156,1112952
EC00345=-798156,1112952
EC00346=-798156,1112952
EC00347=-798156,1112952
EC00348=-798156,1112952
EC00349=-798156,1112952
EC00350=-798156,1112952
EC00351=-798156,1112952
EC00352=-798156,1112952
EC00353=-798156,1112952
EC00354=-798156,1112952
EC00355=-798156,1112952
EC00356=-798156,1112952
EC00357=-798156,1112952
EC00358=-798156,1112952
EC00359=-798156,1112952
EC00360=-798156,1112952
EC00361=-798156,1112952
EC00362=-798156,1112952
EC00363=-798156,1112952
EC00364=-798156,1112952
EC00365=-798156,1112952
EC00366=-798156,1112952
EC00367=-798156,1112952
EC00368=-798156,1112952
EC00369=-798155,1112953
EC00370=798157,1112953
EC00371=798157,1112953
EC00372=798157,1112953
EC00373=798157,1112953
EC00374=798157,1112953
EC00375=798153,1112950
EC00376=798153,1112950
EC00377=798153,1112950
EC00378=798153,1112950
EC00379=798153,1112950
EC00380=798153,1112950
EC00381=798153,1112950
EC00382=798153,1112950
EC00383=798153,1112950
EC00384=798153,1112950
EC00385=798153,1112950
EC00386=798153,1112950
EC00387=798153,1112950
EC00388=798153,1112950
EC00389=798153,1112950
EC00390=798153,1112950
EC00391=798153,1112950
EC00392=798153,1112950
EC00393=798153,1112950
EC00394=798153,1112950
EC00395=798153,1112950
EC00396=798153,1112950
EC00397=798153,1112950
EC00398=798153,1112950
EC00399=798153,1112950
EC00400=798153,1112950
EC00401=798153,1112950
EC00402=798153,1112950
EC00403=798153,1112950
EC00404=798153,1112950
EC00405=798153,1112950
EC00406=798153,1112950
EC00407=798153,1112950
EC00408=798153,1112950
EC00409=798153,1112950
EC00410=798153,1112950
EC00411=798153,1112950
EC00412=798153,1112950
EC00413=798153,1112950
EC00414=798153,1112950
EC00415=798153,1112950
EC00416=798153,1112950
EC00417=798153,1112950
EC00418=798153,1112950
EC00419=798153,1112950
EC00420=798153,1112950
EC00421=798153,1112950
EC00422=798153,1112950
EC00423=798153,1112950
EC00424=798153,1112950
EC00425=798153,1112950
EC00426=798153,1112950
EC00427=798153,1112950
EC00428=798153,1112950
EC00429=798153,1112950
EC00430=798153,1112950
EC00431=798153,1112950
EC00432=798152,1112949
EC00433=798152,1112949
EC00434=798152,1112949
EC00435=798152,1112949
EC00436=798152,1112949
EC00437=798152,1112949
EC00438=798152,1112949
EC00439=798152,1112949
EC00440=798152,1112949
EC00441=798152,1112949
EC00442=798152,1112949
EC00443=798152,1112949
EC00444=798152,1112949
EC00445=798152,1112949
EC00446=798152,1112949
EC00447=798152,1112949
EC00448=798152,1112949
EC00449=798152,1112949
EC00450=798152,1112949
EC00451=798152,1112949
EC00452=798152,1112949
EC00453=798152,1112949
EC00454=798152,1112949
EC00455=798152,1112949
EC00456=798152,1112949
EC00457=798152,1112949
EC00458=798152,1112949
EC00459=798153,1112950
EC00460=798152,1112949
EC00461=798152,1112949
EC00462=798152,1112949
EC00463=798152,1112949
EC00464=798152,1112949
EC00465=798152,1112949
EC00466=798152,1112949
EC00467=798152,1112949
EC00468=798152,1112949
EC00469=798152,1112949
EC00470=798152,1112949
EC00471=798152,1112949
EC00472=798152,1112949
EC00473=798152,1112949
EC00474=798152,1112949
EC00475=798152,1112949
EC00476=798151,1112949
EC00477=798151,1112949
EC00478=798151,1112949
EC00479=798151,1112949
EC00480=798151,1112949
EC00481=798151,1112949
EC00482=798151,1112949
EC00483=798151,1112949
EC00484=798151,1112949
EC00485=798151,1112949
EC00486=798151,1112949
EC00487=798149,1112949
EC00488=798149,1112949
EC00489=798149,1112949
EC00490=798149,1112949
EC00491=798149,1112949
EC00492=798149,1112949
EC00493=798149,1112949
EC00494=798149,1112949
EC00495=798149,1112949
EC00496=798149,1112949
EC00497=798149,1112949
EC00498=798149,1112949
EC00499=798149,1112949
EC00500=798149,1112949
EC00501=798149,1112949
EC00502=798149,1112949
EC00503=798149,1112949
EC00504=798149,1112949
EC00505=798149,1112949
EC00506=798149,1112949
EC00507=798149,1112949
EC00508=798149,1112949
EC00509=798149,1112949
EC00510=798149,1112949
EC00511=798149,1112949
EC00512=798149,1112949
EC00513=798149,1112949
EC00514=798149,1112949
EC00515=798149,1112949
EC00516=798149,1112949
EC00517=798149,1112949
EC00518=798149,1112949
EC00519=798148,1112948
EC00520=798148,1112948
EC00521=798148,1112948
EC00522=798148,1112948
EC00523=798132,1112946
EC00524=798132,1112946
EC00525=798132,1112946
EC00526=798149,1112949
EC00527=798148,1112948
EC00528=798148,1112948
EC00529=798148,1112948
EC00530=798148,1112948
EC00531=798148,1112948
EC00532=798148,1112948
///POSTYPE BASE
///RECTAN
///RCONF 0,0,0,0,0,0,0,0,0,0,0,0,0,0,0,0,0,0,0,0,0,0,0,0
P00006=1.195,-1.322,-3.236,0.0000,0.0000,0.0000
P00021=1.195,-1.322,-3.236,0.0000,0.0000,0.0000
P00022=0.222,-3.123,-1.508,0.0000,0.0000,0.0000
P00023=0.143,-0.036,0.682,0.0000,0.0000,0.0000
P00024=0.145,-0.552,1.326,0.0000,0.0000,0.0000
P00025=-2.003,0.006,0.728,0.0000,0.0000,0.0000
P00026=0.562,-0.002,-0.337,0.0000,0.0000,0.0000
P00027=-0.746,0.015,-9.096,0.0000,0.0000,0.0000
P00028=-2.237,-0.018,-7.702,0.0000,0.0000,0.0000
P00029=-2.156,-0.086,-4.681,0.0000,0.0000,0.0000
P00030=5.926,-4.294,-1.390,0.0000,0.0000,0.0000
P00031=1.853,-0.001,-1.549,0.0000,0.0000,0.0000
P00032=1.957,0.503,-7.217,0.0000,0.0000,0.0000
//INST
///DATE 2025/01/29 14:55
///ATTR SC,RW
///GROUP1 RB1,BS1
///GROUP2 ST1
NOP
MOVJ C00000 BC00000 VJ=100.00  +MOVJ EC00000 VJ=100.00
MOVJ C00001 BC00001 VJ=100.00  +MOVJ EC00001 VJ=100.00
MOVJ C00002 BC00002 VJ=100.00  +MOVJ EC00002 VJ=100.00
SMOVL C00003 BC00003 V=833.3  +MOVJ EC00003
SMOVL C00004 BC00004 V=166.7  +MOVJ EC00004
SREFP 3 C00005 BC00005  +REFP EC00005
CALL JOB:SEARCH-R1-S13D
SET P021 P006
SFTON3D P021
SMOVL C00006 BC00006 V=166.7  +MOVJ EC00006
SREFP 3 C00007 BC00007  +REFP EC00007
CALL JOB:SEARCH-R1-S13D
SET P021 P006
SFTON3D P021
SMOVL C00008 BC00008 V=166.7  +MOVJ EC00008
SFTOF3D
SMOVL C00009 BC00009 V=833.3  +MOVJ EC00009
SMOVL C00010 BC00010 V=166.7  +MOVJ EC00010
SREFP 3 C00011 BC00011  +REFP EC00011
CALL JOB:SEARCH-R1-S13D
SET P022 P006
SFTON3D P022
SMOVL C00012 BC00012 V=166.7  +MOVJ EC00012
SREFP 3 C00013 BC00013  +REFP EC00013
CALL JOB:SEARCH-R1-S13D
SET P022 P006
SFTON3D P022
SMOVL C00014 BC00014 V=166.7  +MOVJ EC00014
SMOVL C00015 BC00015 V=166.7  +MOVJ EC00015
SREFP 3 C00016 BC00016  +REFP EC00016
CALL JOB:SEARCH-R1-S13D
SET P022 P006
SFTON3D P022
SMOVL C00017 BC00017 V=166.7  +MOVJ EC00017
SFTOF3D
SMOVL C00018 BC00018 V=500.0  +MOVJ EC00018
SMOVL C00019 BC00019 V=500.0  +MOVJ EC00019
SMOVL C00020 BC00020 V=166.7  +MOVJ EC00020
SREFP 3 C00021 BC00021  +REFP EC00021
CALL JOB:SEARCH-R1-S13D
SET P023 P006
SFTON3D P023
SMOVL C00022 BC00022 V=166.7  +MOVJ EC00022
SREFP 3 C00023 BC00023  +REFP EC00023
CALL JOB:SEARCH-R1-S13D
SET P023 P006
SFTON3D P023
SMOVL C00024 BC00024 V=166.7  +MOVJ EC00024
SMOVL C00025 BC00025 V=166.7  +MOVJ EC00025
SREFP 3 C00026 BC00026  +REFP EC00026
CALL JOB:SEARCH-R1-S13D
SET P023 P006
SFTON3D P023
SMOVL C00027 BC00027 V=166.7  +MOVJ EC00027
SFTOF3D
SMOVL C00028 BC00028 V=333.3  +MOVJ EC00028
SMOVL C00029 BC00029 V=166.7  +MOVJ EC00029
SREFP 3 C00030 BC00030  +REFP EC00030
CALL JOB:SEARCH-R1-S13D
SET P024 P006
SFTON3D P024
SMOVL C00031 BC00031 V=166.7  +MOVJ EC00031
SREFP 3 C00032 BC00032  +REFP EC00032
CALL JOB:SEARCH-R1-S13D
SET P024 P006
SFTON3D P024
SMOVL C00033 BC00033 V=166.7  +MOVJ EC00033
SMOVL C00034 BC00034 V=166.7  +MOVJ EC00034
SREFP 3 C00035 BC00035  +REFP EC00035
CALL JOB:SEARCH-R1-S13D
SET P024 P006
SFTON3D P024
SMOVL C00036 BC00036 V=166.7  +MOVJ EC00036
SFTOF3D
SMOVL C00037 BC00037 V=333.3  +MOVJ EC00037
SMOVL C00038 BC00038 V=166.7  +MOVJ EC00038
SREFP 3 C00039 BC00039  +REFP EC00039
CALL JOB:SEARCH-R1-S13D
SET P025 P006
SFTON3D P025
SMOVL C00040 BC00040 V=166.7  +MOVJ EC00040
SREFP 3 C00041 BC00041  +REFP EC00041
CALL JOB:SEARCH-R1-S13D
SET P025 P006
SFTON3D P025
SMOVL C00042 BC00042 V=166.7  +MOVJ EC00042
SREFP 3 C00043 BC00043  +REFP EC00043
CALL JOB:SEARCH-R1-S13D
SET P025 P006
SFTON3D P025
SMOVL C00044 BC00044 V=166.7  +MOVJ EC00044
SFTOF3D
SMOVL C00045 BC00045 V=333.3  +MOVJ EC00045
SMOVL C00046 BC00046 V=1000.0  +MOVJ EC00046
SMOVL C00047 BC00047 V=1000.0  +MOVJ EC00047
SMOVL C00048 BC00048 V=1000.0  +MOVJ EC00048
SMOVL C00049 BC00049 V=666.7  +MOVJ EC00049
SMOVL C00050 BC00050 V=666.7  +MOVJ EC00050
SMOVL C00051 BC00051 V=166.7  +MOVJ EC00051
SREFP 3 C00052 BC00052  +REFP EC00052
CALL JOB:SEARCH-R1-S13D
SET P027 P006
SFTON3D P027
SMOVL C00053 BC00053 V=166.7  +MOVJ EC00053
SREFP 3 C00054 BC00054  +REFP EC00054
CALL JOB:SEARCH-R1-S13D
SET P027 P006
SFTON3D P027
SMOVL C00055 BC00055 V=166.7  +MOVJ EC00055
SMOVL C00056 BC00056 V=250.0  +MOVJ EC00056
SMOVL C00057 BC00057 V=250.0  +MOVJ EC00057
SREFP 3 C00058 BC00058  +REFP EC00058
CALL JOB:SEARCH-R1-S13D
SET P027 P006
SFTON3D P027
SMOVL C00059 BC00059 V=166.7  +MOVJ EC00059
SFTOF3D
SMOVL C00060 BC00060 V=250.0  +MOVJ EC00060
SMOVL C00061 BC00061 V=166.7  +MOVJ EC00061
SREFP 3 C00062 BC00062  +REFP EC00062
CALL JOB:SEARCH-R1-S13D
SET P026 P006
SFTON3D P026
SMOVL C00063 BC00063 V=166.7  +MOVJ EC00063
SMOVL C00064 BC00064 V=166.7  +MOVJ EC00064
SREFP 3 C00065 BC00065  +REFP EC00065
CALL JOB:SEARCH-R1-S13D
SET P026 P006
SFTON3D P026
SMOVL C00066 BC00066 V=166.7  +MOVJ EC00066
MACRO1 MJ#(0) ARGF9
SMOVL C00067 BC00067 V=250.0  +MOVJ EC00067
ARCON
SMOVL C00068 BC00068 V=10.0  +MOVJ EC00068
SMOVL C00069 BC00069 V=10.0  +MOVJ EC00069
SFTON3D P027
SMOVL C00070 BC00070 V=10.0  +MOVJ EC00070
ARCOF
SMOVL C00071 BC00071 V=10.0  +MOVJ EC00071
ARCON
SMOVL C00072 BC00072 V=10.0  +MOVJ EC00072
ARCOF
SFTOF3D
SMOVL C00073 BC00073 V=250.0  +MOVJ EC00073
SMOVL C00074 BC00074 V=666.7  +MOVJ EC00074
SMOVL C00075 BC00075 V=666.7  +MOVJ EC00075
SMOVL C00076 BC00076 V=1000.0  +MOVJ EC00076
SMOVL C00077 BC00077 V=1000.0  +MOVJ EC00077
SFTON3D P021
SMOVL C00078 BC00078 V=166.7  +MOVJ EC00078
ARCON
SMOVL C00079 BC00079 V=10.0  +MOVJ EC00079
SFTON3D P022
SMOVL C00080 BC00080 V=10.0  +MOVJ EC00080
SMOVL C00081 BC00081 V=10.0  +MOVJ EC00081
SMOVL C00082 BC00082 V=10.0  +MOVJ EC00082
SMOVL C00083 BC00083 V=10.0  +MOVJ EC00083
SMOVL C00084 BC00084 V=10.0  +MOVJ EC00084
SMOVL C00085 BC00085 V=10.0  +MOVJ EC00085
SFTON3D P023
SMOVL C00086 BC00086 V=10.0  +MOVJ EC00086
SMOVL C00087 BC00087 V=10.0  +MOVJ EC00087
SMOVL C00088 BC00088 V=10.0  +MOVJ EC00088
SMOVL C00089 BC00089 V=10.0  +MOVJ EC00089
SFTON3D P024
SMOVL C00090 BC00090 V=10.0  +MOVJ EC00090
SMOVL C00091 BC00091 V=10.0  +MOVJ EC00091
ARCOF
SFTOF3D
SMOVL C00092 BC00092 V=250.0  +MOVJ EC00092
SMOVL C00093 BC00093 V=500.0  +MOVJ EC00093
SFTON3D P026
SMOVL C00094 BC00094 V=166.7 PL=0  +MOVJ EC00094
ARCON
SMOVL C00095 BC00095 V=10.0  +MOVJ EC00095
SMOVL C00096 BC00096 V=10.0  +MOVJ EC00096
SFTON3D P025
SMOVL C00097 BC00097 V=10.0  +MOVJ EC00097
ARCOF
SFTOF3D
SMOVL C00098 BC00098 V=400.0  +MOVJ EC00098
SFTON3D P024
SMOVL C00099 BC00099 V=166.7  +MOVJ EC00099
ARCON
SMOVL C00100 BC00100 V=10.0  +MOVJ EC00100
SMOVL C00101 BC00101 V=10.0  +MOVJ EC00101
SFTON3D P025
SMOVL C00102 BC00102 V=10.0  +MOVJ EC00102
SMOVL C00103 BC00103 V=10.0  +MOVJ EC00103
ARCOF
SFTOF3D
SMOVL C00104 BC00104 V=250.0  +MOVJ EC00104
SMOVL C00105 BC00105 V=833.3  +MOVJ EC00105
MOVJ C00106 BC00106 VJ=100.00  +MOVJ EC00106 VJ=100.00
MOVJ C00107 BC00107 VJ=100.00  +MOVJ EC00107 VJ=100.00
CALL JOB:CLEAN-R1_KM_NEW
MOVJ C00108 BC00108 VJ=100.00  +MOVJ EC00108 VJ=100.00
MOVJ C00109 BC00109 VJ=100.00  +MOVJ EC00109 VJ=100.00
MOVJ C00110 BC00110 VJ=100.00  +MOVJ EC00110 VJ=100.00
'obrot
MOVJ C00111 BC00111 VJ=100.00  +MOVJ EC00111 VJ=100.00
MOVJ C00112 BC00112 VJ=100.00  +MOVJ EC00112 VJ=100.00
MOVJ C00113 BC00113 VJ=100.00  +MOVJ EC00113 VJ=100.00
SFTOF3D
SMOVL C00114 BC00114 V=500.0  +MOVJ EC00114
SMOVL C00115 BC00115 V=166.7  +MOVJ EC00115
SREFP 3 C00116 BC00116  +REFP EC00116
CALL JOB:SEARCH-R1-S13D
SET P030 P006
SFTON3D P030
SMOVL C00117 BC00117 V=166.7  +MOVJ EC00117
SREFP 3 C00118 BC00118  +REFP EC00118
CALL JOB:SEARCH-R1-S13D
SET P030 P006
SFTON3D P030
SMOVL C00119 BC00119 V=166.7  +MOVJ EC00119
SFTOF3D
SMOVL C00120 BC00120 V=500.0  +MOVJ EC00120
SMOVL C00121 BC00121 V=166.7  +MOVJ EC00121
SREFP 3 C00122 BC00122  +REFP EC00122
CALL JOB:SEARCH-R1-S13D
SET P031 P006
SFTON3D P031
SMOVL C00123 BC00123 V=166.7  +MOVJ EC00123
SREFP 3 C00124 BC00124  +REFP EC00124
CALL JOB:SEARCH-R1-S13D
SET P031 P006
SFTON3D P031
SMOVL C00125 BC00125 V=166.7  +MOVJ EC00125
SMOVL C00126 BC00126 V=416.7  +MOVJ EC00126
'Path S4271
SFTOF3D
MOVJ C00127 BC00127 VJ=50.00  +MOVJ EC00127 VJ=50.00
SMOVL C00128 BC00128 V=166.7  +MOVJ EC00128
SREFP 3 C00129 BC00129  +REFP EC00129
CALL JOB:SEARCH-R1-S13D
SET P021 P006
SFTON3D P021
SMOVL C00130 BC00130 V=166.7  +MOVJ EC00130
SREFP 3 C00131 BC00131  +REFP EC00131
CALL JOB:SEARCH-R1-S13D
SET P021 P006
SFTON3D P021
SMOVL C00132 BC00132 V=166.7  +MOVJ EC00132
SFTOF3D
SMOVL C00133 BC00133 V=833.3  +MOVJ EC00133
SMOVL C00134 BC00134 V=166.7  +MOVJ EC00134
SREFP 3 C00135 BC00135  +REFP EC00135
CALL JOB:SEARCH-R1-S13D
SET P022 P006
SFTON3D P022
SMOVL C00136 BC00136 V=166.7  +MOVJ EC00136
SREFP 3 C00137 BC00137  +REFP EC00137
CALL JOB:SEARCH-R1-S13D
SET P022 P006
SFTON3D P022
SMOVL C00138 BC00138 V=166.7  +MOVJ EC00138
SMOVL C00139 BC00139 V=166.7  +MOVJ EC00139
SMOVL C00140 BC00140 V=166.7  +MOVJ EC00140
SREFP 3 C00141 BC00141  +REFP EC00141
CALL JOB:SEARCH-R1-S13D
SET P022 P006
SFTON3D P022
SMOVL C00142 BC00142 V=166.7  +MOVJ EC00142
SFTOF3D
SMOVL C00143 BC00143 V=500.0  +MOVJ EC00143
SMOVL C00144 BC00144 V=500.0  +MOVJ EC00144
SMOVL C00145 BC00145 V=166.7  +MOVJ EC00145
SREFP 3 C00146 BC00146  +REFP EC00146
CALL JOB:SEARCH-R1-S13D
SET P023 P006
SFTON3D P023
SMOVL C00147 BC00147 V=166.7  +MOVJ EC00147
SREFP 3 C00148 BC00148  +REFP EC00148
CALL JOB:SEARCH-R1-S13D
SET P023 P006
SFTON3D P023
SMOVL C00149 BC00149 V=166.7  +MOVJ EC00149
SMOVL C00150 BC00150 V=166.7  +MOVJ EC00150
SREFP 3 C00151 BC00151  +REFP EC00151
CALL JOB:SEARCH-R1-S13D
SET P023 P006
SFTON3D P023
SMOVL C00152 BC00152 V=166.7  +MOVJ EC00152
SFTOF3D
SMOVL C00153 BC00153 V=333.3  +MOVJ EC00153
SMOVL C00154 BC00154 V=166.7  +MOVJ EC00154
SREFP 3 C00155 BC00155  +REFP EC00155
CALL JOB:SEARCH-R1-S13D
SET P024 P006
SFTON3D P024
SMOVL C00156 BC00156 V=166.7  +MOVJ EC00156
SREFP 3 C00157 BC00157  +REFP EC00157
CALL JOB:SEARCH-R1-S13D
SET P024 P006
SFTON3D P024
SMOVL C00158 BC00158 V=166.7  +MOVJ EC00158
SMOVL C00159 BC00159 V=166.7  +MOVJ EC00159
SREFP 3 C00160 BC00160  +REFP EC00160
CALL JOB:SEARCH-R1-S13D
SET P024 P006
SFTON3D P024
SMOVL C00161 BC00161 V=166.7  +MOVJ EC00161
SFTOF3D
SMOVL C00162 BC00162 V=333.3  +MOVJ EC00162
SMOVL C00163 BC00163 V=333.3  +MOVJ EC00163
SMOVL C00164 BC00164 V=166.7  +MOVJ EC00164
SREFP 3 C00165 BC00165  +REFP EC00165
CALL JOB:SEARCH-R1-S13D
SET P025 P006
SFTON3D P025
SMOVL C00166 BC00166 V=166.7  +MOVJ EC00166
SREFP 3 C00167 BC00167  +REFP EC00167
CALL JOB:SEARCH-R1-S13D
SET P025 P006
SFTON3D P025
SMOVL C00168 BC00168 V=166.7  +MOVJ EC00168
SMOVL C00169 BC00169 V=166.7  +MOVJ EC00169
SREFP 3 C00170 BC00170  +REFP EC00170
CALL JOB:SEARCH-R1-S13D
SET P025 P006
SFTON3D P025
SMOVL C00171 BC00171 V=166.7  +MOVJ EC00171
SFTOF3D
SMOVL C00172 BC00172 V=333.3  +MOVJ EC00172
SMOVL C00173 BC00173 V=1000.0  +MOVJ EC00173
SMOVL C00174 BC00174 V=166.7  +MOVJ EC00174
SMOVL C00175 BC00175 V=166.7  +MOVJ EC00175
SREFP 3 C00176 BC00176  +REFP EC00176
CALL JOB:SEARCH-R1-S13D
SET P027 P006
SFTON3D P027
SMOVL C00177 BC00177 V=166.7  +MOVJ EC00177
SREFP 3 C00178 BC00178  +REFP EC00178
CALL JOB:SEARCH-R1-S13D
SET P027 P006
SFTON3D P027
SMOVL C00179 BC00179 V=166.7  +MOVJ EC00179
SMOVL C00180 BC00180 V=250.0  +MOVJ EC00180
SMOVL C00181 BC00181 V=250.0  +MOVJ EC00181
SREFP 3 C00182 BC00182  +REFP EC00182
CALL JOB:SEARCH-R1-S13D
SET P027 P006
SFTON3D P027
SMOVL C00183 BC00183 V=166.7  +MOVJ EC00183
SFTOF3D
SMOVL C00184 BC00184 V=250.0  +MOVJ EC00184
SMOVL C00185 BC00185 V=166.7  +MOVJ EC00185
SREFP 3 C00186 BC00186  +REFP EC00186
CALL JOB:SEARCH-R1-S13D
SET P026 P006
SFTON3D P026
SMOVL C00187 BC00187 V=166.7  +MOVJ EC00187
SREFP 3 C00188 BC00188  +REFP EC00188
CALL JOB:SEARCH-R1-S13D
SET P026 P006
SFTON3D P026
SMOVL C00189 BC00189 V=166.7  +MOVJ EC00189
SMOVL C00190 BC00190 V=166.7  +MOVJ EC00190
SFTOF3D
SMOVL C00191 BC00191 V=500.0  +MOVJ EC00191
SMOVL C00192 BC00192 V=500.0  +MOVJ EC00192
MOVJ C00193 BC00193 VJ=20.00  +MOVJ EC00193 VJ=20.00
MOVJ C00194 BC00194 VJ=20.00  +MOVJ EC00194 VJ=100.00
MOVJ C00195 BC00195 VJ=20.00  +MOVJ EC00195 VJ=20.00
MACRO1 MJ#(0) ARGF9
SFTON3D P026
SMOVL C00196 BC00196 V=250.0  +MOVJ EC00196
ARCON
SMOVL C00197 BC00197 V=10.0  +MOVJ EC00197
SMOVL C00198 BC00198 V=10.0  +MOVJ EC00198
SFTON3D P027
SMOVL C00199 BC00199 V=10.0  +MOVJ EC00199
SMOVL C00200 BC00200 V=10.0  +MOVJ EC00200
SMOVL C00201 BC00201 V=10.0  +MOVJ EC00201
SMOVL C00202 BC00202 V=10.0  +MOVJ EC00202
ARCOF
SFTOF3D
SMOVL C00203 BC00203 V=250.0  +MOVJ EC00203
SMOVL C00204 BC00204 V=500.0  +MOVJ EC00204
SMOVL C00205 BC00205 V=666.7  +MOVJ EC00205
SMOVL C00206 BC00206 V=500.0  +MOVJ EC00206
MOVJ C00207 BC00207 VJ=20.00  +MOVJ EC00207 VJ=20.00
MOVJ C00208 BC00208 VJ=20.00  +MOVJ EC00208 VJ=20.00
SFTON3D P021
SMOVL C00209 BC00209 V=166.7  +MOVJ EC00209
ARCON
SMOVL C00210 BC00210 V=10.0  +MOVJ EC00210
SFTON3D P022
SMOVL C00211 BC00211 V=10.0  +MOVJ EC00211
SMOVL C00212 BC00212 V=10.0  +MOVJ EC00212
SMOVL C00213 BC00213 V=10.0  +MOVJ EC00213
SMOVL C00214 BC00214 V=10.0  +MOVJ EC00214
SMOVL C00215 BC00215 V=10.0  +MOVJ EC00215
SMOVL C00216 BC00216 V=10.0  +MOVJ EC00216
SFTON3D P023
SMOVL C00217 BC00217 V=10.0  +MOVJ EC00217
SMOVL C00218 BC00218 V=10.0  +MOVJ EC00218
SMOVL C00219 BC00219 V=10.0  +MOVJ EC00219
SMOVL C00220 BC00220 V=10.0  +MOVJ EC00220
SFTON3D P024
SMOVL C00221 BC00221 V=10.0  +MOVJ EC00221
SMOVL C00222 BC00222 V=10.0  +MOVJ EC00222
ARCOF
SFTOF3D
SMOVL C00223 BC00223 V=250.0  +MOVJ EC00223
SMOVL C00224 BC00224 V=500.0  +MOVJ EC00224
SFTON3D P026
SMOVL C00225 BC00225 V=250.0  +MOVJ EC00225
ARCON
SMOVL C00226 BC00226 V=10.0  +MOVJ EC00226
SMOVL C00227 BC00227 V=10.0  +MOVJ EC00227
SFTON3D P025
SMOVL C00228 BC00228 V=10.0  +MOVJ EC00228
ARCOF
SFTOF3D
SMOVL C00229 BC00229 V=400.0  +MOVJ EC00229
SMOVL C00230 BC00230 V=500.0  +MOVJ EC00230
SFTON3D P024
SMOVL C00231 BC00231 V=166.7  +MOVJ EC00231
ARCON
SMOVL C00232 BC00232 V=10.0  +MOVJ EC00232
SMOVL C00233 BC00233 V=10.0  +MOVJ EC00233
SFTON3D P025
SMOVL C00234 BC00234 V=10.0  +MOVJ EC00234
SMOVL C00235 BC00235 V=10.0  +MOVJ EC00235
ARCOF
SFTOF3D
SMOVL C00236 BC00236 V=250.0  +MOVJ EC00236
SMOVL C00237 BC00237 V=416.7  +MOVJ EC00237
SMOVL C00238 BC00238 V=416.7  +MOVJ EC00238
MACRO1 MJ#(0) ARGF14
SFTON3D P030
SMOVL C00239 BC00239 V=166.7  +MOVJ EC00239
ARCON
SFTON3D P031
SMOVL C00240 BC00240 V=10.0  +MOVJ EC00240
SMOVL C00241 BC00241 V=10.0  +MOVJ EC00241
ARCOF
SMOVL C00242 BC00242 V=250.0  +MOVJ EC00242
SFTOF3D
SMOVL C00243 BC00243 V=416.7  +MOVJ EC00243
SMOVL C00244 BC00244 V=833.3  +MOVJ EC00244
MOVJ C00245 BC00245 VJ=100.00  +MOVJ EC00245 VJ=100.00
MOVJ C00246 BC00246 VJ=100.00  +MOVJ EC00246 VJ=100.00
'obrot
MOVJ C00247 BC00247 VJ=100.00  +MOVJ EC00247 VJ=100.00
MOVJ C00248 BC00248 VJ=100.00  +MOVJ EC00248 VJ=100.00
'
MOVJ C00249 BC00249 VJ=100.00  +MOVJ EC00249 VJ=100.00
'DOD. SPOINY WZM. HARDOX
MOVJ C00250 BC00250 VJ=100.00  +MOVJ EC00250 VJ=20.00
MOVJ C00251 BC00251 VJ=100.00  +MOVJ EC00251 VJ=100.00
MOVJ C00252 BC00252 VJ=100.00  +MOVJ EC00252 VJ=100.00
CALL JOB:CLEAN-R1_KM_3P
MOVJ C00253 BC00253 VJ=100.00  +MOVJ EC00253 VJ=100.00
MOVJ C00254 BC00254 VJ=100.00  +MOVJ EC00254 VJ=100.00
MOVJ C00255 BC00255 VJ=100.00  +MOVJ EC00255 VJ=100.00
MOVL C00256 BC00256 V=666.7  +MOVJ EC00256 VJ=100.00
SMOVL C00257 BC00257 V=666.7  +MOVJ EC00257
SMOVL C00258 BC00258 V=166.7  +MOVJ EC00258
SREFP 3 C00259 BC00259  +REFP EC00259
CALL JOB:SEARCH-R1-S13D
SET P021 P006
SFTON3D P021
SMOVL C00260 BC00260 V=166.7  +MOVJ EC00260
SREFP 3 C00261 BC00261  +REFP EC00261
CALL JOB:SEARCH-R1-S13D
SET P021 P006
SFTON3D P021
SMOVL C00262 BC00262 V=166.7  +MOVJ EC00262
SREFP 3 C00263 BC00263  +REFP EC00263
CALL JOB:SEARCH-R1-S13D
SET P021 P006
SFTON3D P021
SMOVL C00264 BC00264 V=166.7  +MOVJ EC00264
SMOVL C00265 BC00265 V=666.7  +MOVJ EC00265
SMOVL C00266 BC00266 V=166.7  +MOVJ EC00266
SREFP 3 C00267 BC00267  +REFP EC00267
CALL JOB:SEARCH-R1-S13D
SET P022 P006
SFTON3D P022
SMOVL C00268 BC00268 V=166.7  +MOVJ EC00268
SREFP 3 C00269 BC00269  +REFP EC00269
CALL JOB:SEARCH-R1-S13D
SET P022 P006
SFTON3D P022
SMOVL C00270 BC00270 V=166.7  +MOVJ EC00270
SREFP 3 C00271 BC00271  +REFP EC00271
CALL JOB:SEARCH-R1-S13D
SET P022 P006
SFTON3D P022
SMOVL C00272 BC00272 V=166.7  +MOVJ EC00272
SMOVL C00273 BC00273 V=666.7  +MOVJ EC00273
SMOVL C00274 BC00274 V=166.7  +MOVJ EC00274
SREFP 3 C00275 BC00275  +REFP EC00275
CALL JOB:SEARCH-R1-S13D
SET P024 P006
SFTON3D P024
SMOVL C00276 BC00276 V=166.7  +MOVJ EC00276
SREFP 3 C00277 BC00277  +REFP EC00277
CALL JOB:SEARCH-R1-S13D
SET P024 P006
SFTON3D P024
SMOVL C00278 BC00278 V=166.7  +MOVJ EC00278
SMOVL C00279 BC00279 V=666.7  +MOVJ EC00279
SMOVL C00280 BC00280 V=166.7  +MOVJ EC00280
SREFP 3 C00281 BC00281  +REFP EC00281
CALL JOB:SEARCH-R1-S13D
SET P023 P006
SFTON3D P023
SMOVL C00282 BC00282 V=166.7  +MOVJ EC00282
SREFP 3 C00283 BC00283  +REFP EC00283
CALL JOB:SEARCH-R1-S13D
SET P023 P006
SFTON3D P023
SMOVL C00284 BC00284 V=166.7  +MOVJ EC00284
SFTOF3D
SMOVL C00285 BC00285 V=666.7  +MOVJ EC00285
SMOVL C00286 BC00286 V=166.7  +MOVJ EC00286
SREFP 3 C00287 BC00287  +REFP EC00287
CALL JOB:SEARCH-R1-S13D
SET P025 P006
SFTON3D P025
SMOVL C00288 BC00288 V=166.7  +MOVJ EC00288
SMOVL C00289 BC00289 V=166.7  +MOVJ EC00289
SMOVL C00290 BC00290 V=166.7  +MOVJ EC00290
SREFP 3 C00291 BC00291  +REFP EC00291
CALL JOB:SEARCH-R1-S13D
SET P025 P006
SFTON3D P025
SMOVL C00292 BC00292 V=166.7  +MOVJ EC00292
SFTOF3D
SMOVL C00293 BC00293 V=666.7  +MOVJ EC00293
SMOVL C00294 BC00294 V=166.7  +MOVJ EC00294
SREFP 3 C00295 BC00295  +REFP EC00295
CALL JOB:SEARCH-R1-S13D
SET P026 P006
SFTON3D P026
SMOVL C00296 BC00296 V=166.7  +MOVJ EC00296
SMOVL C00297 BC00297 V=166.7  +MOVJ EC00297
SMOVL C00298 BC00298 V=166.7  +MOVJ EC00298
SREFP 3 C00299 BC00299  +REFP EC00299
CALL JOB:SEARCH-R1-S13D
SET P026 P006
SFTON3D P026
SMOVL C00300 BC00300 V=166.7  +MOVJ EC00300
SREFP 3 C00301 BC00301  +REFP EC00301
CALL JOB:SEARCH-R1-S13D
SET P026 P006
SFTON3D P026
SMOVL C00302 BC00302 V=166.7  +MOVJ EC00302
SFTOF3D
SMOVL C00303 BC00303 V=666.7  +MOVJ EC00303
SMOVL C00304 BC00304 V=166.7  +MOVJ EC00304
SREFP 3 C00305 BC00305  +REFP EC00305
CALL JOB:SEARCH-R1-S13D
SET P027 P006
SFTON3D P027
SMOVL C00306 BC00306 V=166.7  +MOVJ EC00306
SMOVL C00307 BC00307 V=166.7  +MOVJ EC00307
SMOVL C00308 BC00308 V=166.7  +MOVJ EC00308
SREFP 3 C00309 BC00309  +REFP EC00309
CALL JOB:SEARCH-R1-S13D
SET P027 P006
SFTON3D P027
SMOVL C00310 BC00310 V=166.7  +MOVJ EC00310
SFTOF3D
SMOVL C00311 BC00311 V=666.7  +MOVJ EC00311
SMOVL C00312 BC00312 V=166.7  +MOVJ EC00312
SREFP 3 C00313 BC00313  +REFP EC00313
CALL JOB:SEARCH-R1-S13D
SET P028 P006
SFTON3D P028
SMOVL C00314 BC00314 V=166.7  +MOVJ EC00314
SMOVL C00315 BC00315 V=166.7  +MOVJ EC00315
SMOVL C00316 BC00316 V=166.7  +MOVJ EC00316
SREFP 3 C00317 BC00317  +REFP EC00317
CALL JOB:SEARCH-R1-S13D
SET P028 P006
SFTON3D P028
SMOVL C00318 BC00318 V=166.7  +MOVJ EC00318
SFTOF3D
MOVL C00319 BC00319 V=666.7  +MOVJ EC00319 VJ=100.00
SFTON3D P022
MOVL C00320 BC00320 V=666.7  +MOVJ EC00320 VJ=100.00
MACRO1 MJ#(0) ARGF9
SMOVL C00321 BC00321 V=166.7 PL=0  +MOVJ EC00321
ARCON
SFTON3D P021
SMOVL C00322 BC00322 V=11.7  +MOVJ EC00322
SMOVC C00323 BC00323 V=15.0  +MOVJ EC00323
SMOVC C00324 BC00324 V=15.0  +MOVJ EC00324
SMOVC C00325 BC00325 V=15.0  +MOVJ EC00325
SFTON3D P022
SMOVL C00326 BC00326 V=11.7  +MOVJ EC00326
SMOVL C00327 BC00327 V=11.7  +MOVJ EC00327
SMOVC C00328 BC00328 V=15.0  +MOVJ EC00328
SMOVC C00329 BC00329 V=15.0  +MOVJ EC00329
SMOVC C00330 BC00330 V=15.0  +MOVJ EC00330
ARCOF
SMOVL C00331 BC00331 V=333.3  +MOVJ EC00331
SFTOF3D
SMOVL C00332 BC00332 V=666.7  +MOVJ EC00332
SMOVL C00333 BC00333 V=166.7  +MOVJ EC00333
SFTON3D P024
SMOVL C00334 BC00334 V=166.7 PL=0  +MOVJ EC00334
SWVON WEV#(70)
ARCON
SMOVL C00335 BC00335 V=6.7  +MOVJ EC00335
ARCOF
SWVOF
SMOVL C00336 BC00336 V=166.7  +MOVJ EC00336
SMOVL C00337 BC00337 V=166.7  +MOVJ EC00337
SMOVL C00338 BC00338 V=166.7 PL=0  +MOVJ EC00338
ARCON
SWVON WEV#(70)
SMOVL C00339 BC00339 V=8.3  +MOVJ EC00339
SFTON3D P023
SMOVL C00340 BC00340 V=6.7  +MOVJ EC00340
ARCOF
SWVOF
SMOVL C00341 BC00341 V=166.7  +MOVJ EC00341
SMOVL C00342 BC00342 V=166.7  +MOVJ EC00342
SMOVL C00343 BC00343 V=166.7 PL=0  +MOVJ EC00343
ARCON
SWVON WEV#(70)
SMOVL C00344 BC00344 V=8.3  +MOVJ EC00344
SMOVL C00345 BC00345 V=6.7  +MOVJ EC00345
ARCOF
SWVOF
SMOVL C00346 BC00346 V=166.7  +MOVJ EC00346
SFTOF3D
SMOVL C00347 BC00347 V=666.7  +MOVJ EC00347
SFTON3D P024
SMOVL C00348 BC00348 V=166.7 PL=0  +MOVJ EC00348
ARCON
SMOVL C00349 BC00349 V=15.0  +MOVJ EC00349
SFTON3D P025
SMOVL C00350 BC00350 V=15.0  +MOVJ EC00350
SMOVL C00351 BC00351 V=11.7  +MOVJ EC00351
SFTON3D P026
SMOVL C00352 BC00352 V=11.7  +MOVJ EC00352
SMOVL C00353 BC00353 V=15.0  +MOVJ EC00353
SMOVL C00354 BC00354 V=15.0  +MOVJ EC00354
SMOVL C00355 BC00355 V=15.0  +MOVJ EC00355
SMOVL C00356 BC00356 V=11.7  +MOVJ EC00356
ARCOF
SMOVL C00357 BC00357 V=166.7  +MOVJ EC00357
SFTOF3D
SMOVL C00358 BC00358 V=666.7  +MOVJ EC00358
SMOVL C00359 BC00359 V=666.7  +MOVJ EC00359
SFTON3D P024
SMOVL C00360 BC00360 V=166.7 PL=0  +MOVJ EC00360
ARCON
SMOVL C00361 BC00361 V=15.0  +MOVJ EC00361
SFTON3D P027
SMOVL C00362 BC00362 V=15.0  +MOVJ EC00362
SMOVL C00363 BC00363 V=11.7  +MOVJ EC00363
SFTON3D P028
SMOVL C00364 BC00364 V=11.7  +MOVJ EC00364
SMOVL C00365 BC00365 V=11.7  +MOVJ EC00365
ARCOF
SMOVL C00366 BC00366 V=166.7  +MOVJ EC00366
SFTOF3D
SMOVL C00367 BC00367 V=666.7  +MOVJ EC00367
MOVL C00368 BC00368 V=666.7  +MOVJ EC00368 VJ=0.78
CALL JOB:CLEAN-R1_KM_3P
MOVJ C00369 BC00369 VJ=100.00  +MOVJ EC00369 VJ=100.00
MOVJ C00370 BC00370 VJ=100.00  +MOVJ EC00370 VJ=100.00
MOVJ C00371 BC00371 VJ=100.00  +MOVJ EC00371 VJ=100.00
MOVJ C00372 BC00372 VJ=100.00  +MOVJ EC00372 VJ=100.00
MOVJ C00373 BC00373 VJ=100.00  +MOVJ EC00373 VJ=100.00
MOVJ C00374 BC00374 VJ=100.00  +MOVJ EC00374 VJ=100.00
SMOVL C00375 BC00375 V=666.7  +MOVJ EC00375
SMOVL C00376 BC00376 V=166.7  +MOVJ EC00376
SREFP 3 C00377 BC00377  +REFP EC00377
CALL JOB:SEARCH-R1-S13D
SET P021 P006
SFTON3D P021
SMOVL C00378 BC00378 V=166.7  +MOVJ EC00378
SMOVL C00379 BC00379 V=166.7  +MOVJ EC00379
SMOVL C00380 BC00380 V=166.7  +MOVJ EC00380
SREFP 3 C00381 BC00381  +REFP EC00381
CALL JOB:SEARCH-R1-S13D
SET P021 P006
SFTON3D P021
SMOVL C00382 BC00382 V=166.7  +MOVJ EC00382
SMOVL C00383 BC00383 V=666.7  +MOVJ EC00383
SMOVL C00384 BC00384 V=166.7  +MOVJ EC00384
SREFP 3 C00385 BC00385  +REFP EC00385
CALL JOB:SEARCH-R1-S13D
SET P022 P006
SFTON3D P022
SMOVL C00386 BC00386 V=166.7  +MOVJ EC00386
SREFP 3 C00387 BC00387  +REFP EC00387
CALL JOB:SEARCH-R1-S13D
SET P022 P006
SFTON3D P022
SMOVL C00388 BC00388 V=166.7  +MOVJ EC00388
SREFP 3 C00389 BC00389  +REFP EC00389
CALL JOB:SEARCH-R1-S13D
SET P022 P006
SFTON3D P022
SMOVL C00390 BC00390 V=166.7  +MOVJ EC00390
SMOVL C00391 BC00391 V=666.7  +MOVJ EC00391
SMOVL C00392 BC00392 V=166.7  +MOVJ EC00392
SREFP 3 C00393 BC00393  +REFP EC00393
CALL JOB:SEARCH-R1-S13D
SET P023 P006
SFTON3D P023
SMOVL C00394 BC00394 V=166.7  +MOVJ EC00394
SREFP 3 C00395 BC00395  +REFP EC00395
CALL JOB:SEARCH-R1-S13D
SET P023 P006
SFTON3D P023
SMOVL C00396 BC00396 V=166.7  +MOVJ EC00396
SREFP 3 C00397 BC00397  +REFP EC00397
CALL JOB:SEARCH-R1-S13D
SET P023 P006
SFTON3D P023
SMOVL C00398 BC00398 V=166.7  +MOVJ EC00398
SMOVL C00399 BC00399 V=666.7  +MOVJ EC00399
SMOVL C00400 BC00400 V=166.7  +MOVJ EC00400
SREFP 3 C00401 BC00401  +REFP EC00401
CALL JOB:SEARCH-R1-S13D
SET P024 P006
SFTON3D P024
SMOVL C00402 BC00402 V=166.7  +MOVJ EC00402
SREFP 3 C00403 BC00403  +REFP EC00403
CALL JOB:SEARCH-R1-S13D
SET P024 P006
SFTON3D P024
SMOVL C00404 BC00404 V=166.7  +MOVJ EC00404
SMOVL C00405 BC00405 V=666.7  +MOVJ EC00405
SMOVL C00406 BC00406 V=166.7  +MOVJ EC00406
SREFP 3 C00407 BC00407  +REFP EC00407
CALL JOB:SEARCH-R1-S13D
SET P025 P006
SFTON3D P025
SMOVL C00408 BC00408 V=166.7  +MOVJ EC00408
SREFP 3 C00409 BC00409  +REFP EC00409
CALL JOB:SEARCH-R1-S13D
SET P025 P006
SFTON3D P025
SMOVL C00410 BC00410 V=166.7  +MOVJ EC00410
SMOVL C00411 BC00411 V=666.7  +MOVJ EC00411
SMOVL C00412 BC00412 V=166.7  +MOVJ EC00412
SREFP 3 C00413 BC00413  +REFP EC00413
CALL JOB:SEARCH-R1-S13D
SET P026 P006
SFTON3D P026
SMOVL C00414 BC00414 V=166.7  +MOVJ EC00414
SREFP 3 C00415 BC00415  +REFP EC00415
CALL JOB:SEARCH-R1-S13D
SET P026 P006
SFTON3D P026
SMOVL C00416 BC00416 V=166.7  +MOVJ EC00416
SMOVL C00417 BC00417 V=166.7  +MOVJ EC00417
SREFP 3 C00418 BC00418  +REFP EC00418
CALL JOB:SEARCH-R1-S13D
SET P027 P006
SFTON3D P027
SMOVL C00419 BC00419 V=166.7  +MOVJ EC00419
SREFP 3 C00420 BC00420  +REFP EC00420
CALL JOB:SEARCH-R1-S13D
SET P027 P006
SFTON3D P027
SMOVL C00421 BC00421 V=166.7  +MOVJ EC00421
SMOVL C00422 BC00422 V=166.7  +MOVJ EC00422
SREFP 3 C00423 BC00423  +REFP EC00423
CALL JOB:SEARCH-R1-S13D
SET P028 P006
SFTON3D P028
SMOVL C00424 BC00424 V=166.7  +MOVJ EC00424
SMOVL C00425 BC00425 V=166.7  +MOVJ EC00425
SMOVL C00426 BC00426 V=166.7  +MOVJ EC00426
SREFP 3 C00427 BC00427  +REFP EC00427
CALL JOB:SEARCH-R1-S13D
SET P028 P006
SFTON3D P028
SMOVL C00428 BC00428 V=166.7  +MOVJ EC00428
SFTOF3D
SMOVL C00429 BC00429 V=666.7  +MOVJ EC00429
SFTON3D P022
SMOVL C00430 BC00430 V=666.7  +MOVJ EC00430
SMOVL C00431 BC00431 V=166.7  +MOVJ EC00431
SREFP 3 C00432 BC00432  +REFP EC00432
CALL JOB:SEARCH-R1-S13D
SET P030 P006
SFTON3D P030
SMOVL C00433 BC00433 V=166.7  +MOVJ EC00433
SREFP 3 C00434 BC00434  +REFP EC00434
CALL JOB:SEARCH-R1-S13D
SET P030 P006
SFTON3D P030
SMOVL C00435 BC00435 V=166.7  +MOVJ EC00435
SMOVL C00436 BC00436 V=666.7  +MOVJ EC00436
SMOVL C00437 BC00437 V=166.7  +MOVJ EC00437
SREFP 3 C00438 BC00438  +REFP EC00438
CALL JOB:SEARCH-R1-S13D
SET P029 P006
SFTON3D P029
SMOVL C00439 BC00439 V=166.7  +MOVJ EC00439
SREFP 3 C00440 BC00440  +REFP EC00440
CALL JOB:SEARCH-R1-S13D
SET P029 P006
SFTON3D P029
SMOVL C00441 BC00441 V=166.7  +MOVJ EC00441
SFTOF3D
SMOVL C00442 BC00442 V=166.7  +MOVJ EC00442
SREFP 3 C00443 BC00443  +REFP EC00443
CALL JOB:SEARCH-R1-S13D
SET P031 P006
SFTON3D P031
SMOVL C00444 BC00444 V=166.7  +MOVJ EC00444
SMOVL C00445 BC00445 V=166.7  +MOVJ EC00445
SMOVL C00446 BC00446 V=166.7  +MOVJ EC00446
SREFP 3 C00447 BC00447  +REFP EC00447
CALL JOB:SEARCH-R1-S13D
SET P031 P006
SFTON3D P031
SMOVL C00448 BC00448 V=166.7  +MOVJ EC00448
SMOVL C00449 BC00449 V=666.7  +MOVJ EC00449
SMOVL C00450 BC00450 V=166.7  +MOVJ EC00450
SREFP 3 C00451 BC00451  +REFP EC00451
CALL JOB:SEARCH-R1-S13D
SET P032 P006
SFTON3D P032
SMOVL C00452 BC00452 V=166.7  +MOVJ EC00452
SMOVL C00453 BC00453 V=166.7  +MOVJ EC00453
SMOVL C00454 BC00454 V=166.7  +MOVJ EC00454
SREFP 3 C00455 BC00455  +REFP EC00455
CALL JOB:SEARCH-R1-S13D
SET P032 P006
SFTON3D P032
SMOVL C00456 BC00456 V=166.7  +MOVJ EC00456
SREFP 3 C00457 BC00457  +REFP EC00457
CALL JOB:SEARCH-R1-S13D
SET P032 P006
SFTON3D P032
SMOVL C00458 BC00458 V=166.7  +MOVJ EC00458
SFTOF3D
SMOVL C00459 BC00459 V=666.7  +MOVJ EC00459
MACRO1 MJ#(0) ARGF9
SFTON3D P022
SMOVL C00460 BC00460 V=166.7 PL=0  +MOVJ EC00460
ARCON
SFTON3D P023
SMOVL C00461 BC00461 V=11.7  +MOVJ EC00461
SMOVC C00462 BC00462 V=15.0  +MOVJ EC00462
SMOVC C00463 BC00463 V=15.0  +MOVJ EC00463
SMOVC C00464 BC00464 V=15.0  +MOVJ EC00464
SFTON3D P022
SMOVL C00465 BC00465 V=11.7  +MOVJ EC00465
SMOVL C00466 BC00466 V=11.7  +MOVJ EC00466
SMOVC C00467 BC00467 V=15.0  +MOVJ EC00467
SMOVC C00468 BC00468 V=15.0  +MOVJ EC00468
SMOVC C00469 BC00469 V=15.0  +MOVJ EC00469
ARCOF
SMOVL C00470 BC00470 V=166.7  +MOVJ EC00470
SFTOF3D
SMOVL C00471 BC00471 V=666.7  +MOVJ EC00471
SFTON3D P024
SMOVL C00472 BC00472 V=166.7  +MOVJ EC00472
SMOVL C00473 BC00473 V=166.7 PL=0  +MOVJ EC00473
ARCON
SMOVL C00474 BC00474 V=11.7  +MOVJ EC00474
SMOVC C00475 BC00475 V=15.0  +MOVJ EC00475
SMOVC C00476 BC00476 V=15.0  +MOVJ EC00476
SMOVC C00477 BC00477 V=15.0  +MOVJ EC00477
SMOVL C00478 BC00478 V=11.7  +MOVJ EC00478
SFTON3D P025
SMOVL C00479 BC00479 V=11.7  +MOVJ EC00479
SMOVC C00480 BC00480 V=15.0  +MOVJ EC00480
SMOVC C00481 BC00481 V=15.0  +MOVJ EC00481
SFTON3D P026
SMOVC C00482 BC00482 V=15.0  +MOVJ EC00482
SMOVL C00483 BC00483 V=11.7  +MOVJ EC00483
SFTON3D P027
SMOVL C00484 BC00484 V=11.7  +MOVJ EC00484
ARCOF
SMOVL C00485 BC00485 V=166.7  +MOVJ EC00485
SFTOF3D
SMOVL C00486 BC00486 V=666.7  +MOVJ EC00486
SMOVL C00487 BC00487 V=666.7  +MOVJ EC00487
SFTON3D P029
SMOVL C00488 BC00488 V=666.7  +MOVJ EC00488
SMOVL C00489 BC00489 V=166.7 PL=0  +MOVJ EC00489
ARCON
SWVON WEV#(70)
SMOVL C00490 BC00490 V=6.7  +MOVJ EC00490
ARCOF
SWVOF
SMOVL C00491 BC00491 V=166.7  +MOVJ EC00491
SMOVL C00492 BC00492 V=166.7  +MOVJ EC00492
SMOVL C00493 BC00493 V=166.7 PL=0  +MOVJ EC00493
ARCON
SWVON WEV#(70)
SMOVL C00494 BC00494 V=6.7  +MOVJ EC00494
SFTON3D P030
SMOVL C00495 BC00495 V=6.7  +MOVJ EC00495
ARCOF
SWVOF
SMOVL C00496 BC00496 V=166.7  +MOVJ EC00496
SMOVL C00497 BC00497 V=166.7  +MOVJ EC00497
SMOVL C00498 BC00498 V=166.7 PL=0  +MOVJ EC00498
ARCON
SWVON WEV#(70)
SMOVL C00499 BC00499 V=6.7  +MOVJ EC00499
SMOVL C00500 BC00500 V=6.7  +MOVJ EC00500
ARCOF
SWVOF
SMOVL C00501 BC00501 V=166.7  +MOVJ EC00501
SFTOF3D
SMOVL C00502 BC00502 V=666.7  +MOVJ EC00502
SFTON3D P029
SMOVL C00503 BC00503 V=666.7  +MOVJ EC00503
SMOVL C00504 BC00504 V=166.7 PL=0  +MOVJ EC00504
ARCON
SMOVL C00505 BC00505 V=15.0  +MOVJ EC00505
SFTON3D P031
SMOVL C00506 BC00506 V=15.0  +MOVJ EC00506
SMOVL C00507 BC00507 V=15.0  +MOVJ EC00507
SMOVL C00508 BC00508 V=11.7  +MOVJ EC00508
SFTON3D P032
SMOVL C00509 BC00509 V=11.7  +MOVJ EC00509
SMOVL C00510 BC00510 V=15.0  +MOVJ EC00510
SMOVL C00511 BC00511 V=11.7  +MOVJ EC00511
SMOVL C00512 BC00512 V=15.0  +MOVJ EC00512
SMOVL C00513 BC00513 V=11.7  +MOVJ EC00513
ARCOF
SMOVL C00514 BC00514 V=166.7  +MOVJ EC00514
SFTOF3D
SMOVL C00515 BC00515 V=666.7  +MOVJ EC00515
SFTON3D P029
SMOVL C00516 BC00516 V=666.7  +MOVJ EC00516
SMOVL C00517 BC00517 V=166.7 PL=0  +MOVJ EC00517
ARCON
SMOVL C00518 BC00518 V=15.0  +MOVJ EC00518
SFTON3D P021
SMOVL C00519 BC00519 V=15.0  +MOVJ EC00519
SMOVL C00520 BC00520 V=15.0  +MOVJ EC00520
SMOVL C00521 BC00521 V=11.7  +MOVJ EC00521
SFTON3D P028
SMOVL C00522 BC00522 V=11.7  +MOVJ EC00522
SMOVL C00523 BC00523 V=11.7  +MOVJ EC00523
SMOVL C00524 BC00524 V=11.7  +MOVJ EC00524
ARCOF
SMOVL C00525 BC00525 V=166.7  +MOVJ EC00525
SFTOF3D
SMOVL C00526 BC00526 V=666.7  +MOVJ EC00526
SMOVL C00527 BC00527 V=666.7  +MOVJ EC00527
MOVJ C00528 BC00528 VJ=100.00  +MOVJ EC00528 VJ=100.00
MOVJ C00529 BC00529 VJ=100.00  +MOVJ EC00529 VJ=100.00
MOVJ C00530 BC00530 VJ=100.00  +MOVJ EC00530 VJ=100.00
MOVJ C00531 BC00531 VJ=100.00  +MOVJ EC00531 VJ=100.00
MOVJ C00532 BC00532 VJ=100.00  +MOVJ EC00532 VJ=100.00
END
